LIN {X 0,Y 431.332,Z 858.27,A -85,B 0,C 180,E1 -9447.198,E2 -9447.198} C_VEL
LIN {X 0,Y 431.292,Z 859.283,A -85,B 0,C 180,E1 -9448.132,E2 -9448.132} C_VEL
LIN {X 0,Y 431.285,Z 859.901,A -85,B 0,C 180,E1 -9449.066,E2 -9449.066} C_VEL
LIN {X 0,Y 431.288,Z 860.122,A -85,B 0,C 180,E1 -9450,E2 -9450} C_VEL
LIN {X 0,Y 431.282,Z 859.894,A -85,B 0,C 180,E1 -9450.933,E2 -9450.933} C_VEL
LIN {X 0,Y 431.29,Z 859.263,A -85,B 0,C 180,E1 -9451.867,E2 -9451.867} C_VEL
LIN {X 0,Y 431.33,Z 858.237,A -85,B 0,C 180,E1 -9452.801,E2 -9452.801} C_VEL
LIN {X 0,Y 431.278,Z 856.781,A -85,B 0,C 180,E1 -9453.737,E2 -9453.737} C_VEL
LIN {X 0,Y 431.391,Z 853.758,A -85,B 0,C 180,E1 -9455.14,E2 -9455.14} C_VEL
LIN {X 0,Y 431.441,Z 849.653,A -85,B 0,C 180,E1 -9456.547,E2 -9456.547} C_VEL
LIN {X 0,Y 431.694,Z 843.326,A -85,B 0,C 180,E1 -9458.189,E2 -9458.189} C_VEL
LIN {X 0,Y 432.008,Z 836.432,A -85,B 0,C 180,E1 -9459.598,E2 -9459.598} C_VEL
LIN {X 0,Y 432.42,Z 827.793,A -85,B 0,C 180,E1 -9461.009,E2 -9461.009} C_VEL
LIN {X 0,Y 433.025,Z 818.912,A -85,B 0,C 180,E1 -9462.18,E2 -9462.18} C_VEL
LIN {X 0,Y 433.579,Z 808.605,A -85,B 0,C 180,E1 -9463.29,E2 -9463.29} C_VEL
LIN {X 0,Y 434.126,Z 798.41,A -85,B 0,C 180,E1 -9464.173,E2 -9464.173} C_VEL
LIN {X 0,Y 434.759,Z 786.373,A -85,B 0,C 180,E1 -9464.989,E2 -9464.989} C_VEL
LIN {X 0,Y 435.206,Z 773.862,A -85,B 0,C 180,E1 -9465.633,E2 -9465.633} C_VEL
LIN {X 0,Y 433.854,Z 761.171,A -85,B 0,C 180,E1 -9466.148,E2 -9466.148} C_VEL
LIN {X 0,Y 432.655,Z 748.331,A -85,B 0,C 180,E1 -9466.586,E2 -9466.586} C_VEL
LIN {X 0,Y 432.123,Z 743.343,A -85,B 0,C 180,E1 -9466.716,E2 -9466.716} C_VEL
LIN {X 0,Y 432.465,Z 730.123,A -85,B 0,C 180,E1 -9469.954,E2 -9469.954} C_VEL
LIN {X 0,Y 432.998,Z 716.144,A -85,B 0,C 180,E1 -9473.431,E2 -9473.431} C_VEL
LIN {X 0,Y 433.549,Z 704.201,A -85,B 0,C 180,E1 -9476.454,E2 -9476.454} C_VEL
LIN {X 0,Y 434.228,Z 691.104,A -85,B 0,C 180,E1 -9479.846,E2 -9479.846} C_VEL
LIN {X 0,Y 434.914,Z 679.886,A -85,B 0,C 180,E1 -9482.828,E2 -9482.828} C_VEL
LIN {X 0,Y 435.597,Z 670.042,A -85,B 0,C 180,E1 -9485.508,E2 -9485.508} C_VEL
LIN {X 0,Y 435.806,Z 664.157,A -85,B 0,C 180,E1 -9487.165,E2 -9487.165} C_VEL
LIN {X 0,Y 433.981,Z 654.686,A -85,B 0,C 180,E1 -9490.069,E2 -9490.069} C_VEL
LIN {X 0,Y 432.337,Z 646.633,A -85,B 0,C 180,E1 -9492.69,E2 -9492.69} C_VEL
LIN {X 0,Y 432.376,Z 646.627,A -85,B 0,C 180,E1 -9495.658,E2 -9495.658} C_VEL
LIN {X 0,Y 432.37,Z 646.63,A -85,B 0,C 180,E1 -9498.391,E2 -9498.391} C_VEL
LIN {X 0,Y 432.35,Z 646.63,A -85,B 0,C 180,E1 -9501.851,E2 -9501.851} C_VEL
LIN {X 0,Y 432.337,Z 646.626,A -85,B 0,C 180,E1 -9505.322,E2 -9505.322} C_VEL
LIN {X 0,Y 432.32,Z 646.63,A -85,B 0,C 180,E1 -9508.654,E2 -9508.654} C_VEL
LIN {X 0,Y 432.377,Z 646.623,A -85,B 0,C 180,E1 -9511.368,E2 -9511.368} C_VEL
LIN {X 0,Y 432.36,Z 646.625,A -85,B 0,C 180,E1 -9513.967,E2 -9513.967} C_VEL
LIN {X 0,Y 432.315,Z 646.632,A -85,B 0,C 180,E1 -9517.035,E2 -9517.035} C_VEL
LIN {X 0,Y 432.382,Z 646.622,A -85,B 0,C 180,E1 -9520.514,E2 -9520.514} C_VEL
LIN {X 0,Y 432.425,Z 646.619,A -85,B 0,C 180,E1 -9523.961,E2 -9523.961} C_VEL
LIN {X 0,Y 432.479,Z 646.612,A -85,B 0,C 180,E1 -9527.804,E2 -9527.804} C_VEL
LIN {X 0,Y 432.487,Z 646.612,A -85,B 0,C 180,E1 -9531.59,E2 -9531.59} C_VEL
LIN {X 0,Y 432.592,Z 646.601,A -85,B 0,C 180,E1 -9534.406,E2 -9534.406} C_VEL
LIN {X 0,Y 432.6,Z 646.601,A -85,B 0,C 180,E1 -9538.138,E2 -9538.138} C_VEL
LIN {X 0,Y 432.728,Z 646.587,A -85,B 0,C 180,E1 -9540,E2 -9540} C_VEL
LIN {X 0,Y 432.628,Z 646.804,A -85,B 0,C 180,E1 -9541.745,E2 -9541.745} C_VEL
LIN {X 0,Y 433.797,Z 653.829,A -85,B 0,C 180,E1 -9543.715,E2 -9543.715} C_VEL
LIN {X 0,Y 434.292,Z 658.876,A -85,B 0,C 180,E1 -9545.106,E2 -9545.106} C_VEL
LIN {X 0,Y 434.227,Z 669.203,A -85,B 0,C 180,E1 -9547.907,E2 -9547.907} C_VEL
LIN {X 0,Y 433.886,Z 681.206,A -85,B 0,C 180,E1 -9551.208,E2 -9551.208} C_VEL
LIN {X 0,Y 433.688,Z 689.494,A -85,B 0,C 180,E1 -9553.518,E2 -9553.518} C_VEL
LIN {X 0,Y 433.356,Z 701.793,A -85,B 0,C 180,E1 -9556.973,E2 -9556.973} C_VEL
LIN {X 0,Y 432.958,Z 714.047,A -85,B 0,C 180,E1 -9560.426,E2 -9560.426} C_VEL
LIN {X 0,Y 432.639,Z 724.66,A -85,B 0,C 180,E1 -9563.452,E2 -9563.452} C_VEL
LIN {X 0,Y 432.569,Z 727.887,A -85,B 0,C 180,E1 -9564.347,E2 -9564.347} C_VEL
LIN {X 0,Y 435.121,Z 741.11,A -85,B 0,C 180,E1 -9564.813,E2 -9564.813} C_VEL
LIN {X 0,Y 436.013,Z 747.455,A -85,B 0,C 180,E1 -9565.096,E2 -9565.096} C_VEL
LIN {X 0,Y 435.532,Z 759.628,A -85,B 0,C 180,E1 -9565.688,E2 -9565.688} C_VEL
LIN {X 0,Y 434.958,Z 770.483,A -85,B 0,C 180,E1 -9566.381,E2 -9566.381} C_VEL
LIN {X 0,Y 434.33,Z 781.467,A -85,B 0,C 180,E1 -9567.274,E2 -9567.274} C_VEL
LIN {X 0,Y 433.618,Z 792.684,A -85,B 0,C 180,E1 -9568.426,E2 -9568.426} C_VEL
LIN {X 0,Y 432.951,Z 802.445,A -85,B 0,C 180,E1 -9569.676,E2 -9569.676} C_VEL
LIN {X 0,Y 432.398,Z 811.473,A -85,B 0,C 180,E1 -9571.131,E2 -9571.131} C_VEL
LIN {X 0,Y 431.992,Z 818.185,A -85,B 0,C 180,E1 -9572.471,E2 -9572.471} C_VEL
LIN {X 0,Y 431.665,Z 823.82,A -85,B 0,C 180,E1 -9573.868,E2 -9573.868} C_VEL
LIN {X 0,Y 431.389,Z 828.739,A -85,B 0,C 180,E1 -9575.456,E2 -9575.456} C_VEL
LIN {X 0,Y 431.212,Z 832.39,A -85,B 0,C 180,E1 -9577.088,E2 -9577.088} C_VEL
LIN {X 0,Y 431.094,Z 834.505,A -85,B 0,C 180,E1 -9578.509,E2 -9578.509} C_VEL
LIN {X 0,Y 431.026,Z 835.696,A -85,B 0,C 180,E1 -9579.974,E2 -9579.974} C_VEL
LIN {X 0,Y 430.985,Z 835.911,A -85,B 0,C 180,E1 -9581.401,E2 -9581.401} C_VEL
LIN {X 0,Y 431.012,Z 834.855,A -85,B 0,C 180,E1 -9583.223,E2 -9583.223} C_VEL
LIN {X 0,Y 431.127,Z 833.155,A -85,B 0,C 180,E1 -9584.504,E2 -9584.504} C_VEL
LIN {X 0,Y 431.238,Z 830.613,A -85,B 0,C 180,E1 -9585.814,E2 -9585.814} C_VEL
LIN {X 0,Y 431.432,Z 827.136,A -85,B 0,C 180,E1 -9587.142,E2 -9587.142} C_VEL
LIN {X 0,Y 431.652,Z 822.558,A -85,B 0,C 180,E1 -9588.5,E2 -9588.5} C_VEL
LIN {X 0,Y 431.99,Z 816.732,A -85,B 0,C 180,E1 -9589.875,E2 -9589.875} C_VEL
LIN {X 0,Y 432.47,Z 809.427,A -85,B 0,C 180,E1 -9591.264,E2 -9591.264} C_VEL
LIN {X 0,Y 432.989,Z 801.184,A -85,B 0,C 180,E1 -9592.533,E2 -9592.533} C_VEL
LIN {X 0,Y 433.608,Z 791.196,A -85,B 0,C 180,E1 -9593.776,E2 -9593.776} C_VEL
LIN {X 0,Y 434.236,Z 781.145,A -85,B 0,C 180,E1 -9594.791,E2 -9594.791} C_VEL
LIN {X 0,Y 434.882,Z 769.922,A -85,B 0,C 180,E1 -9595.695,E2 -9595.695} C_VEL
LIN {X 0,Y 435.548,Z 757.776,A -85,B 0,C 180,E1 -9596.451,E2 -9596.451} C_VEL
LIN {X 0,Y 435.872,Z 746.742,A -85,B 0,C 180,E1 -9596.977,E2 -9596.977} C_VEL
LIN {X 0,Y 433.746,Z 734.023,A -85,B 0,C 180,E1 -9597.492,E2 -9597.492} C_VEL
LIN {X 0,Y 432.461,Z 727.38,A -85,B 0,C 180,E1 -9597.714,E2 -9597.714} C_VEL
LIN {X 0,Y 432.921,Z 715.217,A -85,B 0,C 180,E1 -9601.238,E2 -9601.238} C_VEL
LIN {X 0,Y 433.297,Z 703.777,A -85,B 0,C 180,E1 -9604.544,E2 -9604.544} C_VEL
LIN {X 0,Y 433.675,Z 692.539,A -85,B 0,C 180,E1 -9607.802,E2 -9607.802} C_VEL
LIN {X 0,Y 434.013,Z 682.851,A -85,B 0,C 180,E1 -9610.613,E2 -9610.613} C_VEL
LIN {X 0,Y 434.368,Z 671.056,A -85,B 0,C 180,E1 -9614.035,E2 -9614.035} C_VEL
LIN {X 0,Y 434.561,Z 661.142,A -85,B 0,C 180,E1 -9616.914,E2 -9616.914} C_VEL
LIN {X 0,Y 434.514,Z 659.446,A -85,B 0,C 180,E1 -9617.42,E2 -9617.42} C_VEL
LIN {X 0,Y 433.592,Z 657.241,A -85,B 0,C 180,E1 -9618.132,E2 -9618.132} C_VEL
LIN {X 0,Y 430.211,Z 654.112,A -85,B 0,C 180,E1 -9619.298,E2 -9619.298} C_VEL
LIN {X 0,Y 427.311,Z 651.652,A -85,B 0,C 180,E1 -9620.24,E2 -9620.24} C_VEL
LIN {X 0,Y 425.886,Z 649.565,A -85,B 0,C 180,E1 -9620.965,E2 -9620.965} C_VEL
LIN {X 0,Y 425.67,Z 648.783,A -85,B 0,C 180,E1 -9621.21,E2 -9621.21} C_VEL
LIN {X 0,Y 425.459,Z 647.491,A -85,B 0,C 180,E1 -9621.63,E2 -9621.63} C_VEL
LIN {X 0,Y 425.555,Z 647.481,A -85,B 0,C 180,E1 -9624.314,E2 -9624.314} C_VEL
LIN {X 0,Y 425.577,Z 647.478,A -85,B 0,C 180,E1 -9628.108,E2 -9628.108} C_VEL
LIN {X 0,Y 425.705,Z 647.459,A -85,B 0,C 180,E1 -9630.001,E2 -9630.001} C_VEL
LIN {X 0,Y 425.559,Z 647.477,A -85,B 0,C 180,E1 -9632.84,E2 -9632.84} C_VEL
LIN {X 0,Y 425.528,Z 647.477,A -85,B 0,C 180,E1 -9636.639,E2 -9636.639} C_VEL
LIN {X 0,Y 425.405,Z 647.493,A -85,B 0,C 180,E1 -9639.51,E2 -9639.51} C_VEL
LIN {X 0,Y 425.406,Z 647.497,A -85,B 0,C 180,E1 -9642.911,E2 -9642.911} C_VEL
LIN {X 0,Y 425.363,Z 647.504,A -85,B 0,C 180,E1 -9646.605,E2 -9646.605} C_VEL
LIN {X 0,Y 425.33,Z 647.508,A -85,B 0,C 180,E1 -9649.636,E2 -9649.636} C_VEL
LIN {X 0,Y 425.334,Z 647.574,A -85,B 0,C 180,E1 -9651.996,E2 -9651.996} C_VEL
LIN {X 0,Y 428.652,Z 658.894,A -85,B 0,C 180,E1 -9652.79,E2 -9652.79} C_VEL
LIN {X 0,Y 429.276,Z 661.664,A -85,B 0,C 180,E1 -9653.009,E2 -9653.009} C_VEL
LIN {X 0,Y 428.845,Z 672.85,A -85,B 0,C 180,E1 -9653.875,E2 -9653.875} C_VEL
LIN {X 0,Y 428.275,Z 683.125,A -85,B 0,C 180,E1 -9654.867,E2 -9654.867} C_VEL
LIN {X 0,Y 427.705,Z 693.237,A -85,B 0,C 180,E1 -9656.087,E2 -9656.087} C_VEL
LIN {X 0,Y 427.131,Z 702.284,A -85,B 0,C 180,E1 -9657.433,E2 -9657.433} C_VEL
LIN {X 0,Y 426.579,Z 709.888,A -85,B 0,C 180,E1 -9658.839,E2 -9658.839} C_VEL
LIN {X 0,Y 426.091,Z 716.875,A -85,B 0,C 180,E1 -9660.477,E2 -9660.477} C_VEL
LIN {X 0,Y 425.795,Z 721.556,A -85,B 0,C 180,E1 -9661.883,E2 -9661.883} C_VEL
LIN {X 0,Y 425.508,Z 725.849,A -85,B 0,C 180,E1 -9663.595,E2 -9663.595} C_VEL
LIN {X 0,Y 425.268,Z 728.728,A -85,B 0,C 180,E1 -9665.339,E2 -9665.339} C_VEL
LIN {X 0,Y 425.19,Z 729.934,A -85,B 0,C 180,E1 -9666.516,E2 -9666.516} C_VEL
LIN {X 0,Y 425.178,Z 730.484,A -85,B 0,C 180,E1 -9667.705,E2 -9667.705} C_VEL
LIN {X 0,Y 425.238,Z 730.406,A -85,B 0,C 180,E1 -9669.033,E2 -9669.033} C_VEL
LIN {X 0,Y 425.33,Z 729.404,A -85,B 0,C 180,E1 -9670.528,E2 -9670.528} C_VEL
LIN {X 0,Y 425.479,Z 727.476,A -85,B 0,C 180,E1 -9671.987,E2 -9671.987} C_VEL
LIN {X 0,Y 425.747,Z 724.603,A -85,B 0,C 180,E1 -9673.421,E2 -9673.421} C_VEL
LIN {X 0,Y 426.153,Z 719.68,A -85,B 0,C 180,E1 -9675.166,E2 -9675.166} C_VEL
LIN {X 0,Y 426.643,Z 713.798,A -85,B 0,C 180,E1 -9676.735,E2 -9676.735} C_VEL
LIN {X 0,Y 427.105,Z 707.513,A -85,B 0,C 180,E1 -9678.061,E2 -9678.061} C_VEL
LIN {X 0,Y 427.71,Z 699.733,A -85,B 0,C 180,E1 -9679.387,E2 -9679.387} C_VEL
LIN {X 0,Y 428.308,Z 691.12,A -85,B 0,C 180,E1 -9680.585,E2 -9680.585} C_VEL
LIN {X 0,Y 428.931,Z 681.12,A -85,B 0,C 180,E1 -9681.717,E2 -9681.717} C_VEL
LIN {X 0,Y 429.438,Z 671.625,A -85,B 0,C 180,E1 -9682.589,E2 -9682.589} C_VEL
LIN {X 0,Y 429.657,Z 661.647,A -85,B 0,C 180,E1 -9683.341,E2 -9683.341} C_VEL
LIN {X 0,Y 426.566,Z 651.552,A -85,B 0,C 180,E1 -9684.105,E2 -9684.105} C_VEL
LIN {X 0,Y 425.297,Z 647.508,A -85,B 0,C 180,E1 -9684.371,E2 -9684.371} C_VEL
LIN {X 0,Y 425.282,Z 647.515,A -85,B 0,C 180,E1 -9687.437,E2 -9687.437} C_VEL
LIN {X 0,Y 425.292,Z 647.507,A -85,B 0,C 180,E1 -9690.281,E2 -9690.281} C_VEL
LIN {X 0,Y 425.354,Z 647.499,A -85,B 0,C 180,E1 -9693.506,E2 -9693.506} C_VEL
LIN {X 0,Y 425.285,Z 647.502,A -85,B 0,C 180,E1 -9696.634,E2 -9696.634} C_VEL
LIN {X 0,Y 425.296,Z 647.513,A -85,B 0,C 180,E1 -9699.695,E2 -9699.695} C_VEL
LIN {X 0,Y 425.344,Z 647.499,A -85,B 0,C 180,E1 -9702.698,E2 -9702.698} C_VEL
LIN {X 0,Y 425.352,Z 647.503,A -85,B 0,C 180,E1 -9705.65,E2 -9705.65} C_VEL
LIN {X 0,Y 425.352,Z 647.496,A -85,B 0,C 180,E1 -9708.564,E2 -9708.564} C_VEL
LIN {X 0,Y 425.539,Z 647.472,A -85,B 0,C 180,E1 -9712.408,E2 -9712.408} C_VEL
LIN {X 0,Y 425.555,Z 647.476,A -85,B 0,C 180,E1 -9714.313,E2 -9714.313} C_VEL
LIN {X 0,Y 425.577,Z 647.474,A -85,B 0,C 180,E1 -9718.107,E2 -9718.107} C_VEL
LIN {X 0,Y 425.705,Z 647.455,A -85,B 0,C 180,E1 -9720,E2 -9720} C_VEL
LIN {X 0,Y 425.559,Z 647.472,A -85,B 0,C 180,E1 -9722.84,E2 -9722.84} C_VEL
LIN {X 0,Y 425.532,Z 647.478,A -85,B 0,C 180,E1 -9726.639,E2 -9726.639} C_VEL
LIN {X 0,Y 425.403,Z 647.487,A -85,B 0,C 180,E1 -9729.509,E2 -9729.509} C_VEL
LIN {X 0,Y 425.395,Z 647.49,A -85,B 0,C 180,E1 -9732.904,E2 -9732.904} C_VEL
LIN {X 0,Y 425.363,Z 647.497,A -85,B 0,C 180,E1 -9736.605,E2 -9736.605} C_VEL
LIN {X 0,Y 425.33,Z 647.5,A -85,B 0,C 180,E1 -9739.636,E2 -9739.636} C_VEL
LIN {X 0,Y 425.309,Z 647.502,A -85,B 0,C 180,E1 -9743.365,E2 -9743.365} C_VEL
LIN {X 0,Y 425.349,Z 647.502,A -85,B 0,C 180,E1 -9746.844,E2 -9746.844} C_VEL
LIN {X 0,Y 425.293,Z 647.507,A -85,B 0,C 180,E1 -9749.72,E2 -9749.72} C_VEL
LIN {X 0,Y 425.284,Z 647.511,A -85,B 0,C 180,E1 -9753.048,E2 -9753.048} C_VEL
LIN {X 0,Y 425.284,Z 647.511,A -85,B 0,C 180,E1 -9755.929,E2 -9755.929} C_VEL
LIN {X 0,Y 425.296,Z 647.511,A -85,B 0,C 180,E1 -9759.043,E2 -9759.043} C_VEL
LIN {X 0,Y 425.277,Z 647.51,A -85,B 0,C 180,E1 -9762.653,E2 -9762.653} C_VEL
LIN {X 0,Y 425.264,Z 647.515,A -85,B 0,C 180,E1 -9766.044,E2 -9766.044} C_VEL
LIN {X 0,Y 425.339,Z 647.645,A -85,B 0,C 180,E1 -9767.56,E2 -9767.56} C_VEL
LIN {X 0,Y 427.156,Z 656.735,A -85,B 0,C 180,E1 -9770.651,E2 -9770.651} C_VEL
LIN {X 0,Y 428.474,Z 664.587,A -85,B 0,C 180,E1 -9773.118,E2 -9773.118} C_VEL
LIN {X 0,Y 428.013,Z 671.749,A -85,B 0,C 180,E1 -9775.186,E2 -9775.186} C_VEL
LIN {X 0,Y 427.234,Z 684.05,A -85,B 0,C 180,E1 -9778.579,E2 -9778.579} C_VEL
LIN {X 0,Y 426.511,Z 697.918,A -85,B 0,C 180,E1 -9782.257,E2 -9782.257} C_VEL
LIN {X 0,Y 425.939,Z 711.089,A -85,B 0,C 180,E1 -9785.638,E2 -9785.638} C_VEL
LIN {X 0,Y 425.433,Z 724.268,A -85,B 0,C 180,E1 -9788.942,E2 -9788.942} C_VEL
LIN {X 0,Y 425.109,Z 737.422,A -85,B 0,C 180,E1 -9792.191,E2 -9792.191} C_VEL
LIN {X 0,Y 425.001,Z 740.706,A -85,B 0,C 180,E1 -9792.945,E2 -9792.945} C_VEL
LIN {X 0,Y 426.386,Z 753.802,A -85,B 0,C 180,E1 -9793.347,E2 -9793.347} C_VEL
LIN {X 0,Y 427.922,Z 771.686,A -85,B 0,C 180,E1 -9794.047,E2 -9794.047} C_VEL
LIN {X 0,Y 428.234,Z 776.777,A -85,B 0,C 180,E1 -9794.288,E2 -9794.288} C_VEL
LIN {X 0,Y 427.815,Z 787.707,A -85,B 0,C 180,E1 -9794.883,E2 -9794.883} C_VEL
LIN {X 0,Y 427.112,Z 799.468,A -85,B 0,C 180,E1 -9795.71,E2 -9795.71} C_VEL
LIN {X 0,Y 426.476,Z 811.174,A -85,B 0,C 180,E1 -9796.782,E2 -9796.782} C_VEL
LIN {X 0,Y 425.94,Z 820.608,A -85,B 0,C 180,E1 -9797.855,E2 -9797.855} C_VEL
LIN {X 0,Y 425.369,Z 829.198,A -85,B 0,C 180,E1 -9799.047,E2 -9799.047} C_VEL
LIN {X 0,Y 424.891,Z 837.512,A -85,B 0,C 180,E1 -9800.479,E2 -9800.479} C_VEL
LIN {X 0,Y 424.585,Z 844.19,A -85,B 0,C 180,E1 -9801.911,E2 -9801.911} C_VEL
LIN {X 0,Y 424.378,Z 850.124,A -85,B 0,C 180,E1 -9803.538,E2 -9803.538} C_VEL
LIN {X 0,Y 424.29,Z 854.698,A -85,B 0,C 180,E1 -9805.249,E2 -9805.249} C_VEL
LIN {X 0,Y 424.192,Z 856.61,A -85,B 0,C 180,E1 -9806.2,E2 -9806.2} C_VEL
LIN {X 0,Y 424.228,Z 858.067,A -85,B 0,C 180,E1 -9807.151,E2 -9807.151} C_VEL
LIN {X 0,Y 424.214,Z 859.082,A -85,B 0,C 180,E1 -9808.101,E2 -9808.101} C_VEL
LIN {X 0,Y 424.199,Z 859.701,A -85,B 0,C 180,E1 -9809.05,E2 -9809.05} C_VEL
LIN {X 0,Y 424.198,Z 859.923,A -85,B 0,C 180,E1 -9809.999,E2 -9809.999} C_VEL
LIN {X 0,Y 424.195,Z 859.696,A -85,B 0,C 180,E1 -9810.949,E2 -9810.949} C_VEL
LIN {X 0,Y 424.212,Z 859.066,A -85,B 0,C 180,E1 -9811.898,E2 -9811.898} C_VEL
LIN {X 0,Y 424.226,Z 858.04,A -85,B 0,C 180,E1 -9812.848,E2 -9812.848} C_VEL
LIN {X 0,Y 424.185,Z 856.587,A -85,B 0,C 180,E1 -9813.799,E2 -9813.799} C_VEL
LIN {X 0,Y 424.301,Z 853.567,A -85,B 0,C 180,E1 -9815.226,E2 -9815.226} C_VEL
LIN {X 0,Y 424.359,Z 849.468,A -85,B 0,C 180,E1 -9816.657,E2 -9816.657} C_VEL
LIN {X 0,Y 424.629,Z 843.148,A -85,B 0,C 180,E1 -9818.326,E2 -9818.326} C_VEL
LIN {X 0,Y 424.974,Z 836.256,A -85,B 0,C 180,E1 -9819.759,E2 -9819.759} C_VEL
LIN {X 0,Y 425.426,Z 827.626,A -85,B 0,C 180,E1 -9821.192,E2 -9821.192} C_VEL
LIN {X 0,Y 426.053,Z 818.752,A -85,B 0,C 180,E1 -9822.382,E2 -9822.382} C_VEL
LIN {X 0,Y 426.662,Z 808.119,A -85,B 0,C 180,E1 -9823.544,E2 -9823.544} C_VEL
LIN {X 0,Y 427.315,Z 796.719,A -85,B 0,C 180,E1 -9824.525,E2 -9824.525} C_VEL
LIN {X 0,Y 428.016,Z 784.329,A -85,B 0,C 180,E1 -9825.353,E2 -9825.353} C_VEL
LIN {X 0,Y 428.22,Z 773.834,A -85,B 0,C 180,E1 -9825.894,E2 -9825.894} C_VEL
LIN {X 0,Y 427.029,Z 761.62,A -85,B 0,C 180,E1 -9826.407,E2 -9826.407} C_VEL
LIN {X 0,Y 425.059,Z 742.377,A -85,B 0,C 180,E1 -9826.992,E2 -9826.992} C_VEL
LIN {X 0,Y 425.44,Z 729.173,A -85,B 0,C 180,E1 -9830.298,E2 -9830.298} C_VEL
LIN {X 0,Y 425.896,Z 717.225,A -85,B 0,C 180,E1 -9833.33,E2 -9833.33} C_VEL
LIN {X 0,Y 426.477,Z 705.265,A -85,B 0,C 180,E1 -9836.419,E2 -9836.419} C_VEL
LIN {X 0,Y 427.207,Z 692.269,A -85,B 0,C 180,E1 -9839.843,E2 -9839.843} C_VEL
LIN {X 0,Y 427.898,Z 681.246,A -85,B 0,C 180,E1 -9842.82,E2 -9842.82} C_VEL
LIN {X 0,Y 428.699,Z 670.246,A -85,B 0,C 180,E1 -9845.878,E2 -9845.878} C_VEL
LIN {X 0,Y 428.812,Z 665.206,A -85,B 0,C 180,E1 -9847.329,E2 -9847.329} C_VEL
LIN {X 0,Y 426.954,Z 655.628,A -85,B 0,C 180,E1 -9850.327,E2 -9850.327} C_VEL
LIN {X 0,Y 425.296,Z 647.51,A -85,B 0,C 180,E1 -9853.023,E2 -9853.023} C_VEL
LIN {X 0,Y 425.329,Z 647.508,A -85,B 0,C 180,E1 -9856.638,E2 -9856.638} C_VEL
LIN {X 0,Y 425.309,Z 647.507,A -85,B 0,C 180,E1 -9859.875,E2 -9859.875} C_VEL
LIN {X 0,Y 425.284,Z 647.507,A -85,B 0,C 180,E1 -9862.486,E2 -9862.486} C_VEL
LIN {X 0,Y 425.304,Z 647.504,A -85,B 0,C 180,E1 -9865.817,E2 -9865.817} C_VEL
LIN {X 0,Y 425.296,Z 647.505,A -85,B 0,C 180,E1 -9869.236,E2 -9869.236} C_VEL
LIN {X 0,Y 425.346,Z 647.501,A -85,B 0,C 180,E1 -9872.442,E2 -9872.442} C_VEL
LIN {X 0,Y 425.347,Z 647.505,A -85,B 0,C 180,E1 -9875.602,E2 -9875.602} C_VEL
LIN {X 0,Y 425.288,Z 647.509,A -85,B 0,C 180,E1 -9878.681,E2 -9878.681} C_VEL
LIN {X 0,Y 425.328,Z 647.502,A -85,B 0,C 180,E1 -9881.702,E2 -9881.702} C_VEL
LIN {X 0,Y 425.344,Z 647.502,A -85,B 0,C 180,E1 -9884.67,E2 -9884.67} C_VEL
LIN {X 0,Y 425.427,Z 647.492,A -85,B 0,C 180,E1 -9887.598,E2 -9887.598} C_VEL
LIN {X 0,Y 425.438,Z 647.491,A -85,B 0,C 180,E1 -9891.45,E2 -9891.45} C_VEL
LIN {X 0,Y 425.549,Z 647.479,A -85,B 0,C 180,E1 -9894.313,E2 -9894.313} C_VEL
LIN {X 0,Y 425.57,Z 647.477,A -85,B 0,C 180,E1 -9898.107,E2 -9898.107} C_VEL
LIN {X 0,Y 425.697,Z 647.463,A -85,B 0,C 180,E1 -9900,E2 -9900} C_VEL
LIN {X 0,Y 425.55,Z 647.558,A -85,B 0,C 180,E1 -9901.36,E2 -9901.36} C_VEL
LIN {X 0,Y 426.769,Z 654.365,A -85,B 0,C 180,E1 -9903.304,E2 -9903.304} C_VEL
LIN {X 0,Y 427.351,Z 659.35,A -85,B 0,C 180,E1 -9904.716,E2 -9904.716} C_VEL
LIN {X 0,Y 427.342,Z 669.736,A -85,B 0,C 180,E1 -9907.56,E2 -9907.56} C_VEL
LIN {X 0,Y 426.974,Z 680.051,A -85,B 0,C 180,E1 -9910.431,E2 -9910.431} C_VEL
LIN {X 0,Y 426.809,Z 688.62,A -85,B 0,C 180,E1 -9912.844,E2 -9912.844} C_VEL
LIN {X 0,Y 426.477,Z 699.066,A -85,B 0,C 180,E1 -9915.778,E2 -9915.778} C_VEL
LIN {X 0,Y 426.153,Z 709.567,A -85,B 0,C 180,E1 -9918.759,E2 -9918.759} C_VEL
LIN {X 0,Y 425.82,Z 720.147,A -85,B 0,C 180,E1 -9921.799,E2 -9921.799} C_VEL
LIN {X 0,Y 425.592,Z 727.868,A -85,B 0,C 180,E1 -9924.026,E2 -9924.026} C_VEL
LIN {X 0,Y 428.378,Z 742.541,A -85,B 0,C 180,E1 -9924.587,E2 -9924.587} C_VEL
LIN {X 0,Y 429.178,Z 749.058,A -85,B 0,C 180,E1 -9924.89,E2 -9924.89} C_VEL
LIN {X 0,Y 428.69,Z 760.796,A -85,B 0,C 180,E1 -9925.487,E2 -9925.487} C_VEL
LIN {X 0,Y 428.07,Z 771.625,A -85,B 0,C 180,E1 -9926.205,E2 -9926.205} C_VEL
LIN {X 0,Y 427.389,Z 782.348,A -85,B 0,C 180,E1 -9927.107,E2 -9927.107} C_VEL
LIN {X 0,Y 426.65,Z 793.363,A -85,B 0,C 180,E1 -9928.267,E2 -9928.267} C_VEL
LIN {X 0,Y 425.972,Z 802.787,A -85,B 0,C 180,E1 -9929.503,E2 -9929.503} C_VEL
LIN {X 0,Y 425.447,Z 810.807,A -85,B 0,C 180,E1 -9930.803,E2 -9930.803} C_VEL
LIN {X 0,Y 425.006,Z 817.896,A -85,B 0,C 180,E1 -9932.215,E2 -9932.215} C_VEL
LIN {X 0,Y 424.651,Z 823.543,A -85,B 0,C 180,E1 -9933.611,E2 -9933.611} C_VEL
LIN {X 0,Y 424.305,Z 829.136,A -85,B 0,C 180,E1 -9935.431,E2 -9935.431} C_VEL
LIN {X 0,Y 424.183,Z 831.864,A -85,B 0,C 180,E1 -9936.617,E2 -9936.617} C_VEL
LIN {X 0,Y 424.075,Z 833.895,A -85,B 0,C 180,E1 -9937.82,E2 -9937.82} C_VEL
LIN {X 0,Y 423.95,Z 835.297,A -85,B 0,C 180,E1 -9939.046,E2 -9939.046} C_VEL
LIN {X 0,Y 423.919,Z 836.06,A -85,B 0,C 180,E1 -9940.306,E2 -9940.306} C_VEL
LIN {X 0,Y 423.901,Z 836.045,A -85,B 0,C 180,E1 -9941.75,E2 -9941.75} C_VEL
LIN {X 0,Y 423.911,Z 835.132,A -85,B 0,C 180,E1 -9943.159,E2 -9943.159} C_VEL
LIN {X 0,Y 424.034,Z 833.36,A -85,B 0,C 180,E1 -9944.547,E2 -9944.547} C_VEL
LIN {X 0,Y 424.157,Z 830.768,A -85,B 0,C 180,E1 -9945.901,E2 -9945.901} C_VEL
LIN {X 0,Y 424.358,Z 827.326,A -85,B 0,C 180,E1 -9947.234,E2 -9947.234} C_VEL
LIN {X 0,Y 424.653,Z 822,A -85,B 0,C 180,E1 -9948.812,E2 -9948.812} C_VEL
LIN {X 0,Y 425.074,Z 814.92,A -85,B 0,C 180,E1 -9950.427,E2 -9950.427} C_VEL
LIN {X 0,Y 425.548,Z 807.735,A -85,B 0,C 180,E1 -9951.735,E2 -9951.735} C_VEL
LIN {X 0,Y 426.221,Z 798.161,A -85,B 0,C 180,E1 -9953.146,E2 -9953.146} C_VEL
LIN {X 0,Y 426.953,Z 787.532,A -85,B 0,C 180,E1 -9954.388,E2 -9954.388} C_VEL
LIN {X 0,Y 427.594,Z 777.252,A -85,B 0,C 180,E1 -9955.359,E2 -9955.359} C_VEL
LIN {X 0,Y 428.225,Z 766.551,A -85,B 0,C 180,E1 -9956.169,E2 -9956.169} C_VEL
LIN {X 0,Y 428.837,Z 753.63,A -85,B 0,C 180,E1 -9956.915,E2 -9956.915} C_VEL
LIN {X 0,Y 429.043,Z 747.886,A -85,B 0,C 180,E1 -9957.179,E2 -9957.179} C_VEL
LIN {X 0,Y 426.915,Z 735.03,A -85,B 0,C 180,E1 -9957.726,E2 -9957.726} C_VEL
LIN {X 0,Y 425.485,Z 727.51,A -85,B 0,C 180,E1 -9957.982,E2 -9957.982} C_VEL
LIN {X 0,Y 425.916,Z 715.771,A -85,B 0,C 180,E1 -9961.412,E2 -9961.412} C_VEL
LIN {X 0,Y 426.3,Z 704.802,A -85,B 0,C 180,E1 -9964.62,E2 -9964.62} C_VEL
LIN {X 0,Y 426.672,Z 694.137,A -85,B 0,C 180,E1 -9967.738,E2 -9967.738} C_VEL
LIN {X 0,Y 427.055,Z 683.725,A -85,B 0,C 180,E1 -9970.784,E2 -9970.784} C_VEL
LIN {X 0,Y 427.437,Z 671.868,A -85,B 0,C 180,E1 -9974.259,E2 -9974.259} C_VEL
LIN {X 0,Y 427.626,Z 661.902,A -85,B 0,C 180,E1 -9977.182,E2 -9977.182} C_VEL
LIN {X 0,Y 426.933,Z 655.631,A -85,B 0,C 180,E1 -9979.088,E2 -9979.088} C_VEL
LIN {X 0,Y 425.67,Z 648.783,A -85,B 0,C 180,E1 -9981.21,E2 -9981.21} C_VEL
LIN {X 0,Y 425.132,Z 647.83,A -85,B 0,C 180,E1 -9981.703,E2 -9981.703} C_VEL
LIN {X 0,Y 424.201,Z 647.646,A -85,B 0,C 180,E1 -9982.211,E2 -9982.211} C_VEL
LIN {X 0,Y 419.432,Z 648.323,A -85,B 0,C 180,E1 -9984.292,E2 -9984.292} C_VEL
LIN {X 0,Y 418.42,Z 648.379,A -85,B 0,C 180,E1 -9985.109,E2 -9985.109} C_VEL
LIN {X 0,Y 418.322,Z 648.381,A -85,B 0,C 180,E1 -9985.385,E2 -9985.385} C_VEL
LIN {X 0,Y 418.546,Z 648.353,A -85,B 0,C 180,E1 -9988.076,E2 -9988.076} C_VEL
LIN {X 0,Y 418.674,Z 648.335,A -85,B 0,C 180,E1 -9990.001,E2 -9990.001} C_VEL
LIN {X 0,Y 418.513,Z 648.354,A -85,B 0,C 180,E1 -9992.888,E2 -9992.888} C_VEL
LIN {X 0,Y 418.492,Z 648.353,A -85,B 0,C 180,E1 -9996.752,E2 -9996.752} C_VEL
LIN {X 0,Y 418.361,Z 648.37,A -85,B 0,C 180,E1 -9999.671,E2 -9999.671} C_VEL
LIN {X 0,Y 418.357,Z 648.374,A -85,B 0,C 180,E1 -10003.007,E2 -10003.007} C_VEL
LIN {X 0,Y 418.315,Z 648.381,A -85,B 0,C 180,E1 -10006.736,E2 -10006.736} C_VEL
LIN {X 0,Y 418.284,Z 648.385,A -85,B 0,C 180,E1 -10009.795,E2 -10009.795} C_VEL
LIN {X 0,Y 418.307,Z 648.382,A -85,B 0,C 180,E1 -10011.72,E2 -10011.72} C_VEL
LIN {X 0,Y 421.639,Z 659.821,A -85,B 0,C 180,E1 -10012.543,E2 -10012.543} C_VEL
LIN {X 0,Y 422.388,Z 662.544,A -85,B 0,C 180,E1 -10012.768,E2 -10012.768} C_VEL
LIN {X 0,Y 422.006,Z 673.831,A -85,B 0,C 180,E1 -10013.658,E2 -10013.658} C_VEL
LIN {X 0,Y 421.425,Z 683.885,A -85,B 0,C 180,E1 -10014.641,E2 -10014.641} C_VEL
LIN {X 0,Y 420.841,Z 693.947,A -85,B 0,C 180,E1 -10015.867,E2 -10015.867} C_VEL
LIN {X 0,Y 420.266,Z 702.746,A -85,B 0,C 180,E1 -10017.187,E2 -10017.187} C_VEL
LIN {X 0,Y 419.691,Z 709.946,A -85,B 0,C 180,E1 -10018.506,E2 -10018.506} C_VEL
LIN {X 0,Y 419.304,Z 715.451,A -85,B 0,C 180,E1 -10019.739,E2 -10019.739} C_VEL
LIN {X 0,Y 418.892,Z 721.217,A -85,B 0,C 180,E1 -10021.34,E2 -10021.34} C_VEL
LIN {X 0,Y 418.594,Z 725.495,A -85,B 0,C 180,E1 -10022.915,E2 -10022.915} C_VEL
LIN {X 0,Y 418.298,Z 729.122,A -85,B 0,C 180,E1 -10024.838,E2 -10024.838} C_VEL
LIN {X 0,Y 418.177,Z 730.71,A -85,B 0,C 180,E1 -10026.225,E2 -10026.225} C_VEL
LIN {X 0,Y 418.154,Z 731.535,A -85,B 0,C 180,E1 -10027.82,E2 -10027.82} C_VEL
LIN {X 0,Y 418.246,Z 731.163,A -85,B 0,C 180,E1 -10029.683,E2 -10029.683} C_VEL
LIN {X 0,Y 418.361,Z 730.067,A -85,B 0,C 180,E1 -10030.932,E2 -10030.932} C_VEL
LIN {X 0,Y 418.637,Z 727.035,A -85,B 0,C 180,E1 -10032.876,E2 -10032.876} C_VEL
LIN {X 0,Y 418.953,Z 723.836,A -85,B 0,C 180,E1 -10034.248,E2 -10034.248} C_VEL
LIN {X 0,Y 419.313,Z 719.692,A -85,B 0,C 180,E1 -10035.616,E2 -10035.616} C_VEL
LIN {X 0,Y 419.754,Z 714.49,A -85,B 0,C 180,E1 -10036.977,E2 -10036.977} C_VEL
LIN {X 0,Y 420.326,Z 706.835,A -85,B 0,C 180,E1 -10038.563,E2 -10038.563} C_VEL
LIN {X 0,Y 420.933,Z 699.393,A -85,B 0,C 180,E1 -10039.804,E2 -10039.804} C_VEL
LIN {X 0,Y 421.536,Z 691.319,A -85,B 0,C 180,E1 -10040.916,E2 -10040.916} C_VEL
LIN {X 0,Y 422.173,Z 681.946,A -85,B 0,C 180,E1 -10041.979,E2 -10041.979} C_VEL
LIN {X 0,Y 422.742,Z 671.495,A -85,B 0,C 180,E1 -10042.939,E2 -10042.939} C_VEL
LIN {X 0,Y 423.029,Z 663.901,A -85,B 0,C 180,E1 -10043.513,E2 -10043.513} C_VEL
LIN {X 0,Y 419.591,Z 652.47,A -85,B 0,C 180,E1 -10044.405,E2 -10044.405} C_VEL
LIN {X 0,Y 418.265,Z 648.384,A -85,B 0,C 180,E1 -10044.7,E2 -10044.7} C_VEL
LIN {X 0,Y 418.246,Z 648.392,A -85,B 0,C 180,E1 -10047.472,E2 -10047.472} C_VEL
LIN {X 0,Y 418.269,Z 648.381,A -85,B 0,C 180,E1 -10050.896,E2 -10050.896} C_VEL
LIN {X 0,Y 418.269,Z 648.382,A -85,B 0,C 180,E1 -10054.096,E2 -10054.096} C_VEL
LIN {X 0,Y 418.232,Z 648.381,A -85,B 0,C 180,E1 -10057.264,E2 -10057.264} C_VEL
LIN {X 0,Y 418.284,Z 648.382,A -85,B 0,C 180,E1 -10060.364,E2 -10060.364} C_VEL
LIN {X 0,Y 418.327,Z 648.376,A -85,B 0,C 180,E1 -10063.405,E2 -10063.405} C_VEL
LIN {X 0,Y 418.347,Z 648.372,A -85,B 0,C 180,E1 -10066.999,E2 -10066.999} C_VEL
LIN {X 0,Y 418.342,Z 648.374,A -85,B 0,C 180,E1 -10070.329,E2 -10070.329} C_VEL
LIN {X 0,Y 418.515,Z 648.348,A -85,B 0,C 180,E1 -10072.28,E2 -10072.28} C_VEL
LIN {X 0,Y 418.515,Z 648.354,A -85,B 0,C 180,E1 -10074.217,E2 -10074.217} C_VEL
LIN {X 0,Y 418.546,Z 648.349,A -85,B 0,C 180,E1 -10078.076,E2 -10078.076} C_VEL
LIN {X 0,Y 418.674,Z 648.331,A -85,B 0,C 180,E1 -10080,E2 -10080} C_VEL
LIN {X 0,Y 418.512,Z 648.35,A -85,B 0,C 180,E1 -10082.888,E2 -10082.888} C_VEL
LIN {X 0,Y 418.495,Z 648.353,A -85,B 0,C 180,E1 -10086.751,E2 -10086.751} C_VEL
LIN {X 0,Y 418.402,Z 648.36,A -85,B 0,C 180,E1 -10088.695,E2 -10088.695} C_VEL
LIN {X 0,Y 418.317,Z 648.376,A -85,B 0,C 180,E1 -10091.631,E2 -10091.631} C_VEL
LIN {X 0,Y 418.304,Z 648.38,A -85,B 0,C 180,E1 -10094.597,E2 -10094.597} C_VEL
LIN {X 0,Y 418.289,Z 648.376,A -85,B 0,C 180,E1 -10097.604,E2 -10097.604} C_VEL
LIN {X 0,Y 418.252,Z 648.387,A -85,B 0,C 180,E1 -10100.663,E2 -10100.663} C_VEL
LIN {X 0,Y 418.29,Z 648.377,A -85,B 0,C 180,E1 -10103.781,E2 -10103.781} C_VEL
LIN {X 0,Y 418.312,Z 648.377,A -85,B 0,C 180,E1 -10107.071,E2 -10107.071} C_VEL
LIN {X 0,Y 418.246,Z 648.388,A -85,B 0,C 180,E1 -10110.272,E2 -10110.272} C_VEL
LIN {X 0,Y 418.25,Z 648.385,A -85,B 0,C 180,E1 -10113.677,E2 -10113.677} C_VEL
LIN {X 0,Y 418.242,Z 648.389,A -85,B 0,C 180,E1 -10117.224,E2 -10117.224} C_VEL
LIN {X 0,Y 418.251,Z 648.386,A -85,B 0,C 180,E1 -10119.682,E2 -10119.682} C_VEL
LIN {X 0,Y 418.232,Z 648.391,A -85,B 0,C 180,E1 -10122.321,E2 -10122.321} C_VEL
LIN {X 0,Y 418.238,Z 648.391,A -85,B 0,C 180,E1 -10125.109,E2 -10125.109} C_VEL
LIN {X 0,Y 418.279,Z 648.479,A -85,B 0,C 180,E1 -10127.176,E2 -10127.176} C_VEL
LIN {X 0,Y 420.089,Z 657.482,A -85,B 0,C 180,E1 -10130.316,E2 -10130.316} C_VEL
LIN {X 0,Y 421.435,Z 665.136,A -85,B 0,C 180,E1 -10132.806,E2 -10132.806} C_VEL
LIN {X 0,Y 421.287,Z 670.085,A -85,B 0,C 180,E1 -10134.276,E2 -10134.276} C_VEL
LIN {X 0,Y 420.454,Z 682.022,A -85,B 0,C 180,E1 -10137.663,E2 -10137.663} C_VEL
LIN {X 0,Y 419.704,Z 694.021,A -85,B 0,C 180,E1 -10140.947,E2 -10140.947} C_VEL
LIN {X 0,Y 419.114,Z 706.077,A -85,B 0,C 180,E1 -10144.152,E2 -10144.152} C_VEL
LIN {X 0,Y 418.561,Z 718.859,A -85,B 0,C 180,E1 -10147.443,E2 -10147.443} C_VEL
LIN {X 0,Y 418.144,Z 733.349,A -85,B 0,C 180,E1 -10151.122,E2 -10151.122} C_VEL
LIN {X 0,Y 417.989,Z 739.311,A -85,B 0,C 180,E1 -10152.614,E2 -10152.614} C_VEL
LIN {X 0,Y 419.554,Z 754.545,A -85,B 0,C 180,E1 -10153.118,E2 -10153.118} C_VEL
LIN {X 0,Y 421.033,Z 772.305,A -85,B 0,C 180,E1 -10153.826,E2 -10153.826} C_VEL
LIN {X 0,Y 421.309,Z 778.843,A -85,B 0,C 180,E1 -10154.147,E2 -10154.147} C_VEL
LIN {X 0,Y 420.72,Z 790.99,A -85,B 0,C 180,E1 -10154.87,E2 -10154.87} C_VEL
LIN {X 0,Y 420.072,Z 802.121,A -85,B 0,C 180,E1 -10155.727,E2 -10155.727} C_VEL
LIN {X 0,Y 419.378,Z 813.139,A -85,B 0,C 180,E1 -10156.801,E2 -10156.801} C_VEL
LIN {X 0,Y 418.842,Z 822.152,A -85,B 0,C 180,E1 -10157.892,E2 -10157.892} C_VEL
LIN {X 0,Y 418.149,Z 831.902,A -85,B 0,C 180,E1 -10159.345,E2 -10159.345} C_VEL
LIN {X 0,Y 417.735,Z 839.656,A -85,B 0,C 180,E1 -10160.803,E2 -10160.803} C_VEL
LIN {X 0,Y 417.415,Z 845.844,A -85,B 0,C 180,E1 -10162.259,E2 -10162.259} C_VEL
LIN {X 0,Y 417.266,Z 850.355,A -85,B 0,C 180,E1 -10163.586,E2 -10163.586} C_VEL
LIN {X 0,Y 417.219,Z 854.474,A -85,B 0,C 180,E1 -10165.168,E2 -10165.168} C_VEL
LIN {X 0,Y 417.104,Z 856.39,A -85,B 0,C 180,E1 -10166.135,E2 -10166.135} C_VEL
LIN {X 0,Y 417.125,Z 857.855,A -85,B 0,C 180,E1 -10167.102,E2 -10167.102} C_VEL
LIN {X 0,Y 417.138,Z 858.875,A -85,B 0,C 180,E1 -10168.068,E2 -10168.068} C_VEL
LIN {X 0,Y 417.115,Z 859.497,A -85,B 0,C 180,E1 -10169.034,E2 -10169.034} C_VEL
LIN {X 0,Y 417.112,Z 859.723,A -85,B 0,C 180,E1 -10169.999,E2 -10169.999} C_VEL
LIN {X 0,Y 417.112,Z 859.502,A -85,B 0,C 180,E1 -10170.965,E2 -10170.965} C_VEL
LIN {X 0,Y 417.135,Z 858.874,A -85,B 0,C 180,E1 -10171.931,E2 -10171.931} C_VEL
LIN {X 0,Y 417.122,Z 857.848,A -85,B 0,C 180,E1 -10172.897,E2 -10172.897} C_VEL
LIN {X 0,Y 417.097,Z 856.399,A -85,B 0,C 180,E1 -10173.864,E2 -10173.864} C_VEL
LIN {X 0,Y 417.213,Z 853.382,A -85,B 0,C 180,E1 -10175.315,E2 -10175.315} C_VEL
LIN {X 0,Y 417.276,Z 849.286,A -85,B 0,C 180,E1 -10176.77,E2 -10176.77} C_VEL
LIN {X 0,Y 417.565,Z 842.968,A -85,B 0,C 180,E1 -10178.468,E2 -10178.468} C_VEL
LIN {X 0,Y 417.935,Z 836.079,A -85,B 0,C 180,E1 -10179.925,E2 -10179.925} C_VEL
LIN {X 0,Y 418.347,Z 829.044,A -85,B 0,C 180,E1 -10181.139,E2 -10181.139} C_VEL
LIN {X 0,Y 418.964,Z 820.546,A -85,B 0,C 180,E1 -10182.349,E2 -10182.349} C_VEL
LIN {X 0,Y 419.609,Z 810.041,A -85,B 0,C 180,E1 -10183.561,E2 -10183.561} C_VEL
LIN {X 0,Y 420.24,Z 799.656,A -85,B 0,C 180,E1 -10184.528,E2 -10184.528} C_VEL
LIN {X 0,Y 420.944,Z 788.245,A -85,B 0,C 180,E1 -10185.369,E2 -10185.369} C_VEL
LIN {X 0,Y 421.493,Z 776.479,A -85,B 0,C 180,E1 -10186.031,E2 -10186.031} C_VEL
LIN {X 0,Y 420.329,Z 763.51,A -85,B 0,C 180,E1 -10186.625,E2 -10186.625} C_VEL
LIN {X 0,Y 418.979,Z 750.125,A -85,B 0,C 180,E1 -10187.035,E2 -10187.035} C_VEL
LIN {X 0,Y 418.009,Z 741.364,A -85,B 0,C 180,E1 -10187.285,E2 -10187.285} C_VEL
LIN {X 0,Y 418.405,Z 728.198,A -85,B 0,C 180,E1 -10190.654,E2 -10190.654} C_VEL
LIN {X 0,Y 419.009,Z 714.313,A -85,B 0,C 180,E1 -10194.263,E2 -10194.263} C_VEL
LIN {X 0,Y 419.647,Z 702.352,A -85,B 0,C 180,E1 -10197.425,E2 -10197.425} C_VEL
LIN {X 0,Y 420.412,Z 689.406,A -85,B 0,C 180,E1 -10200.933,E2 -10200.933} C_VEL
LIN {X 0,Y 421.315,Z 677.426,A -85,B 0,C 180,E1 -10204.261,E2 -10204.261} C_VEL
LIN {X 0,Y 421.94,Z 668.17,A -85,B 0,C 180,E1 -10206.917,E2 -10206.917} C_VEL
LIN {X 0,Y 421.293,Z 663.467,A -85,B 0,C 180,E1 -10208.366,E2 -10208.366} C_VEL
LIN {X 0,Y 419.261,Z 653.226,A -85,B 0,C 180,E1 -10211.691,E2 -10211.691} C_VEL
LIN {X 0,Y 418.225,Z 648.39,A -85,B 0,C 180,E1 -10213.388,E2 -10213.388} C_VEL
LIN {X 0,Y 418.281,Z 648.384,A -85,B 0,C 180,E1 -10216.458,E2 -10216.458} C_VEL
LIN {X 0,Y 418.264,Z 648.383,A -85,B 0,C 180,E1 -10219.122,E2 -10219.122} C_VEL
LIN {X 0,Y 418.236,Z 648.385,A -85,B 0,C 180,E1 -10222.164,E2 -10222.164} C_VEL
LIN {X 0,Y 418.262,Z 648.379,A -85,B 0,C 180,E1 -10225.419,E2 -10225.419} C_VEL
LIN {X 0,Y 418.212,Z 648.387,A -85,B 0,C 180,E1 -10228.604,E2 -10228.604} C_VEL
LIN {X 0,Y 418.291,Z 648.38,A -85,B 0,C 180,E1 -10231.936,E2 -10231.936} C_VEL
LIN {X 0,Y 418.285,Z 648.379,A -85,B 0,C 180,E1 -10235.162,E2 -10235.162} C_VEL
LIN {X 0,Y 418.229,Z 648.387,A -85,B 0,C 180,E1 -10238.303,E2 -10238.303} C_VEL
LIN {X 0,Y 418.279,Z 648.384,A -85,B 0,C 180,E1 -10241.383,E2 -10241.383} C_VEL
LIN {X 0,Y 418.298,Z 648.38,A -85,B 0,C 180,E1 -10244.406,E2 -10244.406} C_VEL
LIN {X 0,Y 418.366,Z 648.371,A -85,B 0,C 180,E1 -10247.386,E2 -10247.386} C_VEL
LIN {X 0,Y 418.356,Z 648.374,A -85,B 0,C 180,E1 -10250.329,E2 -10250.329} C_VEL
LIN {X 0,Y 418.488,Z 648.358,A -85,B 0,C 180,E1 -10253.249,E2 -10253.249} C_VEL
LIN {X 0,Y 418.335,Z 648.376,A -85,B 0,C 180,E1 -10255.181,E2 -10255.181} C_VEL
LIN {X 0,Y 418.539,Z 648.353,A -85,B 0,C 180,E1 -10258.075,E2 -10258.075} C_VEL
LIN {X 0,Y 418.667,Z 648.338,A -85,B 0,C 180,E1 -10260,E2 -10260} C_VEL
LIN {X 0,Y 418.531,Z 648.552,A -85,B 0,C 180,E1 -10261.022,E2 -10261.022} C_VEL
LIN {X 0,Y 419.772,Z 654.921,A -85,B 0,C 180,E1 -10262.879,E2 -10262.879} C_VEL
LIN {X 0,Y 420.506,Z 661.635,A -85,B 0,C 180,E1 -10264.793,E2 -10264.793} C_VEL
LIN {X 0,Y 420.417,Z 672.014,A -85,B 0,C 180,E1 -10267.685,E2 -10267.685} C_VEL
LIN {X 0,Y 420.051,Z 684.161,A -85,B 0,C 180,E1 -10271.093,E2 -10271.093} C_VEL
LIN {X 0,Y 419.689,Z 694.481,A -85,B 0,C 180,E1 -10274.069,E2 -10274.069} C_VEL
LIN {X 0,Y 419.372,Z 705.615,A -85,B 0,C 180,E1 -10277.213,E2 -10277.213} C_VEL
LIN {X 0,Y 418.942,Z 717.425,A -85,B 0,C 180,E1 -10280.627,E2 -10280.627} C_VEL
LIN {X 0,Y 418.613,Z 728.081,A -85,B 0,C 180,E1 -10283.729,E2 -10283.729} C_VEL
LIN {X 0,Y 421.329,Z 741.8,A -85,B 0,C 180,E1 -10284.252,E2 -10284.252} C_VEL
LIN {X 0,Y 422.362,Z 750.129,A -85,B 0,C 180,E1 -10284.647,E2 -10284.647} C_VEL
LIN {X 0,Y 421.832,Z 761.954,A -85,B 0,C 180,E1 -10285.273,E2 -10285.273} C_VEL
LIN {X 0,Y 421.125,Z 773.296,A -85,B 0,C 180,E1 -10286.062,E2 -10286.062} C_VEL
LIN {X 0,Y 420.392,Z 784.523,A -85,B 0,C 180,E1 -10287.057,E2 -10287.057} C_VEL
LIN {X 0,Y 419.612,Z 795.161,A -85,B 0,C 180,E1 -10288.239,E2 -10288.239} C_VEL
LIN {X 0,Y 418.954,Z 804.07,A -85,B 0,C 180,E1 -10289.469,E2 -10289.469} C_VEL
LIN {X 0,Y 418.382,Z 812.188,A -85,B 0,C 180,E1 -10290.841,E2 -10290.841} C_VEL
LIN {X 0,Y 417.932,Z 819.043,A -85,B 0,C 180,E1 -10292.27,E2 -10292.27} C_VEL
LIN {X 0,Y 417.531,Z 824.666,A -85,B 0,C 180,E1 -10293.743,E2 -10293.743} C_VEL
LIN {X 0,Y 417.224,Z 829.731,A -85,B 0,C 180,E1 -10295.485,E2 -10295.485} C_VEL
LIN {X 0,Y 417.007,Z 833.506,A -85,B 0,C 180,E1 -10297.353,E2 -10297.353} C_VEL
LIN {X 0,Y 416.846,Z 835.614,A -85,B 0,C 180,E1 -10299.146,E2 -10299.146} C_VEL
LIN {X 0,Y 416.79,Z 836.358,A -85,B 0,C 180,E1 -10301.119,E2 -10301.119} C_VEL
LIN {X 0,Y 416.802,Z 835.924,A -85,B 0,C 180,E1 -10302.413,E2 -10302.413} C_VEL
LIN {X 0,Y 416.857,Z 834.739,A -85,B 0,C 180,E1 -10303.728,E2 -10303.728} C_VEL
LIN {X 0,Y 416.998,Z 832.774,A -85,B 0,C 180,E1 -10305.061,E2 -10305.061} C_VEL
LIN {X 0,Y 417.159,Z 829.929,A -85,B 0,C 180,E1 -10306.422,E2 -10306.422} C_VEL
LIN {X 0,Y 417.412,Z 826.097,A -85,B 0,C 180,E1 -10307.802,E2 -10307.802} C_VEL
LIN {X 0,Y 417.718,Z 819.971,A -85,B 0,C 180,E1 -10309.488,E2 -10309.488} C_VEL
LIN {X 0,Y 418.284,Z 812.344,A -85,B 0,C 180,E1 -10311.116,E2 -10311.116} C_VEL
LIN {X 0,Y 418.798,Z 804.341,A -85,B 0,C 180,E1 -10312.473,E2 -10312.473} C_VEL
LIN {X 0,Y 419.538,Z 794.387,A -85,B 0,C 180,E1 -10313.839,E2 -10313.839} C_VEL
LIN {X 0,Y 420.28,Z 783.531,A -85,B 0,C 180,E1 -10315.023,E2 -10315.023} C_VEL
LIN {X 0,Y 420.976,Z 772.609,A -85,B 0,C 180,E1 -10315.977,E2 -10315.977} C_VEL
LIN {X 0,Y 421.723,Z 760.615,A -85,B 0,C 180,E1 -10316.792,E2 -10316.792} C_VEL
LIN {X 0,Y 422.225,Z 749.476,A -85,B 0,C 180,E1 -10317.368,E2 -10317.368} C_VEL
LIN {X 0,Y 420.367,Z 737.535,A -85,B 0,C 180,E1 -10317.905,E2 -10317.905} C_VEL
LIN {X 0,Y 418.491,Z 727.646,A -85,B 0,C 180,E1 -10318.258,E2 -10318.258} C_VEL
LIN {X 0,Y 418.986,Z 714.993,A -85,B 0,C 180,E1 -10321.988,E2 -10321.988} C_VEL
LIN {X 0,Y 419.44,Z 702.206,A -85,B 0,C 180,E1 -10325.764,E2 -10325.764} C_VEL
LIN {X 0,Y 419.847,Z 691.554,A -85,B 0,C 180,E1 -10328.907,E2 -10328.907} C_VEL
LIN {X 0,Y 420.218,Z 680.991,A -85,B 0,C 180,E1 -10332.028,E2 -10332.028} C_VEL
LIN {X 0,Y 420.632,Z 669.293,A -85,B 0,C 180,E1 -10335.486,E2 -10335.486} C_VEL
LIN {X 0,Y 420.664,Z 662.681,A -85,B 0,C 180,E1 -10337.457,E2 -10337.457} C_VEL
LIN {X 0,Y 419.874,Z 656.416,A -85,B 0,C 180,E1 -10339.391,E2 -10339.391} C_VEL
LIN {X 0,Y 418.461,Z 648.362,A -85,B 0,C 180,E1 -10341.927,E2 -10341.927} C_VEL
LIN {X 0,Y 418.514,Z 648.358,A -85,B 0,C 180,E1 -10344.218,E2 -10344.218} C_VEL
LIN {X 0,Y 418.322,Z 648.381,A -85,B 0,C 180,E1 -10345.385,E2 -10345.385} C_VEL
LIN {X 0,Y 417.617,Z 648.469,A -85,B 0,C 180,E1 -10346.191,E2 -10346.191} C_VEL
LIN {X 0,Y 414.792,Z 648.821,A -85,B 0,C 180,E1 -10347.501,E2 -10347.501} C_VEL
LIN {X 0,Y 412.493,Z 649.107,A -85,B 0,C 180,E1 -10348.559,E2 -10348.559} C_VEL
LIN {X 0,Y 411.594,Z 649.217,A -85,B 0,C 180,E1 -10349.376,E2 -10349.376} C_VEL
LIN {X 0,Y 411.566,Z 649.22,A -85,B 0,C 180,E1 -10349.651,E2 -10349.651} C_VEL
LIN {X 0,Y 411.468,Z 649.232,A -85,B 0,C 180,E1 -10352.938,E2 -10352.938} C_VEL
LIN {X 0,Y 411.455,Z 649.23,A -85,B 0,C 180,E1 -10356.868,E2 -10356.868} C_VEL
LIN {X 0,Y 411.31,Z 649.248,A -85,B 0,C 180,E1 -10359.839,E2 -10359.839} C_VEL
LIN {X 0,Y 411.315,Z 649.251,A -85,B 0,C 180,E1 -10363.11,E2 -10363.11} C_VEL
LIN {X 0,Y 411.259,Z 649.26,A -85,B 0,C 180,E1 -10366.889,E2 -10366.889} C_VEL
LIN {X 0,Y 411.234,Z 649.263,A -85,B 0,C 180,E1 -10369.987,E2 -10369.987} C_VEL
LIN {X 0,Y 411.248,Z 649.324,A -85,B 0,C 180,E1 -10371.458,E2 -10371.458} C_VEL
LIN {X 0,Y 414.626,Z 660.729,A -85,B 0,C 180,E1 -10372.288,E2 -10372.288} C_VEL
LIN {X 0,Y 415.622,Z 664.786,A -85,B 0,C 180,E1 -10372.625,E2 -10372.625} C_VEL
LIN {X 0,Y 415.084,Z 676.343,A -85,B 0,C 180,E1 -10373.575,E2 -10373.575} C_VEL
LIN {X 0,Y 414.466,Z 686.99,A -85,B 0,C 180,E1 -10374.681,E2 -10374.681} C_VEL
LIN {X 0,Y 413.835,Z 696.988,A -85,B 0,C 180,E1 -10375.967,E2 -10375.967} C_VEL
LIN {X 0,Y 413.19,Z 705.567,A -85,B 0,C 180,E1 -10377.339,E2 -10377.339} C_VEL
LIN {X 0,Y 412.601,Z 712.796,A -85,B 0,C 180,E1 -10378.764,E2 -10378.764} C_VEL
LIN {X 0,Y 412.105,Z 719.731,A -85,B 0,C 180,E1 -10380.488,E2 -10380.488} C_VEL
LIN {X 0,Y 411.779,Z 724.253,A -85,B 0,C 180,E1 -10381.944,E2 -10381.944} C_VEL
LIN {X 0,Y 411.446,Z 728.327,A -85,B 0,C 180,E1 -10383.72,E2 -10383.72} C_VEL
LIN {X 0,Y 411.191,Z 731.067,A -85,B 0,C 180,E1 -10385.53,E2 -10385.53} C_VEL
LIN {X 0,Y 411.135,Z 732.127,A -85,B 0,C 180,E1 -10386.748,E2 -10386.748} C_VEL
LIN {X 0,Y 411.158,Z 732.613,A -85,B 0,C 180,E1 -10388.16,E2 -10388.16} C_VEL
LIN {X 0,Y 411.248,Z 732.187,A -85,B 0,C 180,E1 -10389.734,E2 -10389.734} C_VEL
LIN {X 0,Y 411.401,Z 730.806,A -85,B 0,C 180,E1 -10391.266,E2 -10391.266} C_VEL
LIN {X 0,Y 411.668,Z 727.88,A -85,B 0,C 180,E1 -10393.069,E2 -10393.069} C_VEL
LIN {X 0,Y 411.982,Z 724.849,A -85,B 0,C 180,E1 -10394.381,E2 -10394.381} C_VEL
LIN {X 0,Y 412.462,Z 719.724,A -85,B 0,C 180,E1 -10396.047,E2 -10396.047} C_VEL
LIN {X 0,Y 412.974,Z 714.435,A -85,B 0,C 180,E1 -10397.394,E2 -10397.394} C_VEL
LIN {X 0,Y 413.472,Z 707.775,A -85,B 0,C 180,E1 -10398.776,E2 -10398.776} C_VEL
LIN {X 0,Y 414.186,Z 699.469,A -85,B 0,C 180,E1 -10400.167,E2 -10400.167} C_VEL
LIN {X 0,Y 414.862,Z 690.98,A -85,B 0,C 180,E1 -10401.322,E2 -10401.322} C_VEL
LIN {X 0,Y 415.558,Z 680.327,A -85,B 0,C 180,E1 -10402.495,E2 -10402.495} C_VEL
LIN {X 0,Y 416.182,Z 669.221,A -85,B 0,C 180,E1 -10403.469,E2 -10403.469} C_VEL
LIN {X 0,Y 416.181,Z 665.279,A -85,B 0,C 180,E1 -10403.769,E2 -10403.769} C_VEL
LIN {X 0,Y 412.934,Z 654.47,A -85,B 0,C 180,E1 -10404.643,E2 -10404.643} C_VEL
LIN {X 0,Y 411.226,Z 649.261,A -85,B 0,C 180,E1 -10405.042,E2 -10405.042} C_VEL
LIN {X 0,Y 411.166,Z 649.269,A -85,B 0,C 180,E1 -10408.003,E2 -10408.003} C_VEL
LIN {X 0,Y 411.219,Z 649.261,A -85,B 0,C 180,E1 -10411.41,E2 -10411.41} C_VEL
LIN {X 0,Y 411.237,Z 649.256,A -85,B 0,C 180,E1 -10413.619,E2 -10413.619} C_VEL
LIN {X 0,Y 411.196,Z 649.257,A -85,B 0,C 180,E1 -10416.852,E2 -10416.852} C_VEL
LIN {X 0,Y 411.216,Z 649.264,A -85,B 0,C 180,E1 -10420.051,E2 -10420.051} C_VEL
LIN {X 0,Y 411.266,Z 649.254,A -85,B 0,C 180,E1 -10423.131,E2 -10423.131} C_VEL
LIN {X 0,Y 411.307,Z 649.249,A -85,B 0,C 180,E1 -10426.896,E2 -10426.896} C_VEL
LIN {X 0,Y 411.294,Z 649.254,A -85,B 0,C 180,E1 -10430.161,E2 -10430.161} C_VEL
LIN {X 0,Y 411.483,Z 649.224,A -85,B 0,C 180,E1 -10432.147,E2 -10432.147} C_VEL
LIN {X 0,Y 411.477,Z 649.232,A -85,B 0,C 180,E1 -10434.118,E2 -10434.118} C_VEL
LIN {X 0,Y 411.515,Z 649.224,A -85,B 0,C 180,E1 -10438.043,E2 -10438.043} C_VEL
LIN {X 0,Y 411.644,Z 649.206,A -85,B 0,C 180,E1 -10440,E2 -10440} C_VEL
LIN {X 0,Y 411.468,Z 649.227,A -85,B 0,C 180,E1 -10442.937,E2 -10442.937} C_VEL
LIN {X 0,Y 411.462,Z 649.229,A -85,B 0,C 180,E1 -10446.867,E2 -10446.867} C_VEL
LIN {X 0,Y 411.295,Z 649.246,A -85,B 0,C 180,E1 -10449.839,E2 -10449.839} C_VEL
LIN {X 0,Y 411.307,Z 649.243,A -85,B 0,C 180,E1 -10453.104,E2 -10453.104} C_VEL
LIN {X 0,Y 411.259,Z 649.253,A -85,B 0,C 180,E1 -10456.889,E2 -10456.889} C_VEL
LIN {X 0,Y 411.232,Z 649.257,A -85,B 0,C 180,E1 -10459.987,E2 -10459.987} C_VEL
LIN {X 0,Y 411.205,Z 649.259,A -85,B 0,C 180,E1 -10463.148,E2 -10463.148} C_VEL
LIN {X 0,Y 411.24,Z 649.259,A -85,B 0,C 180,E1 -10466.381,E2 -10466.381} C_VEL
LIN {X 0,Y 411.202,Z 649.262,A -85,B 0,C 180,E1 -10469.713,E2 -10469.713} C_VEL
LIN {X 0,Y 411.208,Z 649.264,A -85,B 0,C 180,E1 -10473.156,E2 -10473.156} C_VEL
LIN {X 0,Y 411.195,Z 649.268,A -85,B 0,C 180,E1 -10476.553,E2 -10476.553} C_VEL
LIN {X 0,Y 411.215,Z 649.263,A -85,B 0,C 180,E1 -10479.728,E2 -10479.728} C_VEL
LIN {X 0,Y 411.176,Z 649.263,A -85,B 0,C 180,E1 -10483.134,E2 -10483.134} C_VEL
LIN {X 0,Y 411.21,Z 649.367,A -85,B 0,C 180,E1 -10486.787,E2 -10486.787} C_VEL
LIN {X 0,Y 413.04,Z 658.207,A -85,B 0,C 180,E1 -10489.969,E2 -10489.969} C_VEL
LIN {X 0,Y 414.534,Z 666.842,A -85,B 0,C 180,E1 -10492.829,E2 -10492.829} C_VEL
LIN {X 0,Y 414.236,Z 672.456,A -85,B 0,C 180,E1 -10494.526,E2 -10494.526} C_VEL
LIN {X 0,Y 413.441,Z 683.15,A -85,B 0,C 180,E1 -10497.624,E2 -10497.624} C_VEL
LIN {X 0,Y 412.647,Z 695.104,A -85,B 0,C 180,E1 -10500.961,E2 -10500.961} C_VEL
LIN {X 0,Y 412.051,Z 707.16,A -85,B 0,C 180,E1 -10504.219,E2 -10504.219} C_VEL
LIN {X 0,Y 411.532,Z 718.665,A -85,B 0,C 180,E1 -10507.249,E2 -10507.249} C_VEL
LIN {X 0,Y 411.094,Z 731.437,A -85,B 0,C 180,E1 -10510.561,E2 -10510.561} C_VEL
LIN {X 0,Y 410.947,Z 738.164,A -85,B 0,C 180,E1 -10512.286,E2 -10512.286} C_VEL
LIN {X 0,Y 412.587,Z 753.603,A -85,B 0,C 180,E1 -10512.815,E2 -10512.815} C_VEL
LIN {X 0,Y 413.967,Z 771.802,A -85,B 0,C 180,E1 -10513.542,E2 -10513.542} C_VEL
LIN {X 0,Y 414.436,Z 778.404,A -85,B 0,C 180,E1 -10513.877,E2 -10513.877} C_VEL
LIN {X 0,Y 413.865,Z 790.608,A -85,B 0,C 180,E1 -10514.613,E2 -10514.613} C_VEL
LIN {X 0,Y 413.135,Z 801.887,A -85,B 0,C 180,E1 -10515.493,E2 -10515.493} C_VEL
LIN {X 0,Y 412.449,Z 812.824,A -85,B 0,C 180,E1 -10516.575,E2 -10516.575} C_VEL
LIN {X 0,Y 411.869,Z 821.855,A -85,B 0,C 180,E1 -10517.684,E2 -10517.684} C_VEL
LIN {X 0,Y 411.132,Z 831.621,A -85,B 0,C 180,E1 -10519.161,E2 -10519.161} C_VEL
LIN {X 0,Y 410.68,Z 839.396,A -85,B 0,C 180,E1 -10520.643,E2 -10520.643} C_VEL
LIN {X 0,Y 410.367,Z 845.598,A -85,B 0,C 180,E1 -10522.125,E2 -10522.125} C_VEL
LIN {X 0,Y 410.193,Z 850.447,A -85,B 0,C 180,E1 -10523.587,E2 -10523.587} C_VEL
LIN {X 0,Y 410.148,Z 854.25,A -85,B 0,C 180,E1 -10525.085,E2 -10525.085} C_VEL
LIN {X 0,Y 410.02,Z 856.17,A -85,B 0,C 180,E1 -10526.068,E2 -10526.068} C_VEL
LIN {X 0,Y 410.022,Z 857.643,A -85,B 0,C 180,E1 -10527.052,E2 -10527.052} C_VEL
LIN {X 0,Y 410.063,Z 858.668,A -85,B 0,C 180,E1 -10528.035,E2 -10528.035} C_VEL
LIN {X 0,Y 410.034,Z 859.293,A -85,B 0,C 180,E1 -10529.017,E2 -10529.017} C_VEL
LIN {X 0,Y 410.029,Z 859.523,A -85,B 0,C 180,E1 -10529.999,E2 -10529.999} C_VEL
LIN {X 0,Y 410.031,Z 859.307,A -85,B 0,C 180,E1 -10530.982,E2 -10530.982} C_VEL
LIN {X 0,Y 410.06,Z 858.681,A -85,B 0,C 180,E1 -10531.964,E2 -10531.964} C_VEL
LIN {X 0,Y 410.019,Z 857.656,A -85,B 0,C 180,E1 -10532.947,E2 -10532.947} C_VEL
LIN {X 0,Y 410.013,Z 856.212,A -85,B 0,C 180,E1 -10533.931,E2 -10533.931} C_VEL
LIN {X 0,Y 410.128,Z 853.197,A -85,B 0,C 180,E1 -10535.407,E2 -10535.407} C_VEL
LIN {X 0,Y 410.199,Z 849.105,A -85,B 0,C 180,E1 -10536.888,E2 -10536.888} C_VEL
LIN {X 0,Y 410.527,Z 842.793,A -85,B 0,C 180,E1 -10538.614,E2 -10538.614} C_VEL
LIN {X 0,Y 410.918,Z 835.921,A -85,B 0,C 180,E1 -10540.096,E2 -10540.096} C_VEL
LIN {X 0,Y 411.338,Z 828.906,A -85,B 0,C 180,E1 -10541.331,E2 -10541.331} C_VEL
LIN {X 0,Y 412.007,Z 820.442,A -85,B 0,C 180,E1 -10542.561,E2 -10542.561} C_VEL
LIN {X 0,Y 412.675,Z 809.969,A -85,B 0,C 180,E1 -10543.793,E2 -10543.793} C_VEL
LIN {X 0,Y 413.452,Z 798.19,A -85,B 0,C 180,E1 -10544.897,E2 -10544.897} C_VEL
LIN {X 0,Y 414.221,Z 786.33,A -85,B 0,C 180,E1 -10545.751,E2 -10545.751} C_VEL
LIN {X 0,Y 414.614,Z 776.609,A -85,B 0,C 180,E1 -10546.304,E2 -10546.304} C_VEL
LIN {X 0,Y 413.533,Z 764.139,A -85,B 0,C 180,E1 -10546.894,E2 -10546.894} C_VEL
LIN {X 0,Y 412.268,Z 750.93,A -85,B 0,C 180,E1 -10547.322,E2 -10547.322} C_VEL
LIN {X 0,Y 410.926,Z 740.305,A -85,B 0,C 180,E1 -10547.611,E2 -10547.611} C_VEL
LIN {X 0,Y 411.384,Z 727.243,A -85,B 0,C 180,E1 -10551.023,E2 -10551.023} C_VEL
LIN {X 0,Y 412.052,Z 713.389,A -85,B 0,C 180,E1 -10554.7,E2 -10554.7} C_VEL
LIN {X 0,Y 412.704,Z 701.134,A -85,B 0,C 180,E1 -10558.019,E2 -10558.019} C_VEL
LIN {X 0,Y 413.48,Z 689.531,A -85,B 0,C 180,E1 -10561.225,E2 -10561.225} C_VEL
LIN {X 0,Y 414.513,Z 676.589,A -85,B 0,C 180,E1 -10564.905,E2 -10564.905} C_VEL
LIN {X 0,Y 414.93,Z 668.648,A -85,B 0,C 180,E1 -10567.243,E2 -10567.243} C_VEL
LIN {X 0,Y 413.698,Z 661.629,A -85,B 0,C 180,E1 -10569.488,E2 -10569.488} C_VEL
LIN {X 0,Y 411.734,Z 651.855,A -85,B 0,C 180,E1 -10572.779,E2 -10572.779} C_VEL
LIN {X 0,Y 411.182,Z 649.268,A -85,B 0,C 180,E1 -10573.739,E2 -10573.739} C_VEL
LIN {X 0,Y 411.228,Z 649.262,A -85,B 0,C 180,E1 -10576.873,E2 -10576.873} C_VEL
LIN {X 0,Y 411.226,Z 649.263,A -85,B 0,C 180,E1 -10580.269,E2 -10580.269} C_VEL
LIN {X 0,Y 411.192,Z 649.263,A -85,B 0,C 180,E1 -10583.446,E2 -10583.446} C_VEL
LIN {X 0,Y 411.203,Z 649.262,A -85,B 0,C 180,E1 -10586.873,E2 -10586.873} C_VEL
LIN {X 0,Y 411.237,Z 649.256,A -85,B 0,C 180,E1 -10590.642,E2 -10590.642} C_VEL
LIN {X 0,Y 411.233,Z 649.259,A -85,B 0,C 180,E1 -10593.619,E2 -10593.619} C_VEL
LIN {X 0,Y 411.199,Z 649.262,A -85,B 0,C 180,E1 -10596.852,E2 -10596.852} C_VEL
LIN {X 0,Y 411.21,Z 649.26,A -85,B 0,C 180,E1 -10600.05,E2 -10600.05} C_VEL
LIN {X 0,Y 411.258,Z 649.257,A -85,B 0,C 180,E1 -10603.131,E2 -10603.131} C_VEL
LIN {X 0,Y 411.309,Z 649.25,A -85,B 0,C 180,E1 -10606.89,E2 -10606.89} C_VEL
LIN {X 0,Y 411.304,Z 649.252,A -85,B 0,C 180,E1 -10610.161,E2 -10610.161} C_VEL
LIN {X 0,Y 411.455,Z 649.234,A -85,B 0,C 180,E1 -10613.133,E2 -10613.133} C_VEL
LIN {X 0,Y 411.306,Z 649.253,A -85,B 0,C 180,E1 -10615.099,E2 -10615.099} C_VEL
LIN {X 0,Y 411.508,Z 649.228,A -85,B 0,C 180,E1 -10618.042,E2 -10618.042} C_VEL
LIN {X 0,Y 411.534,Z 649.279,A -85,B 0,C 180,E1 -10620.581,E2 -10620.581} C_VEL
LIN {X 0,Y 413.016,Z 657.177,A -85,B 0,C 180,E1 -10622.926,E2 -10622.926} C_VEL
LIN {X 0,Y 413.672,Z 663.927,A -85,B 0,C 180,E1 -10624.873,E2 -10624.873} C_VEL
LIN {X 0,Y 413.503,Z 674.347,A -85,B 0,C 180,E1 -10627.815,E2 -10627.815} C_VEL
LIN {X 0,Y 413.058,Z 688.236,A -85,B 0,C 180,E1 -10631.781,E2 -10631.781} C_VEL
LIN {X 0,Y 412.7,Z 698.717,A -85,B 0,C 180,E1 -10634.8,E2 -10634.8} C_VEL
LIN {X 0,Y 412.3,Z 709.362,A -85,B 0,C 180,E1 -10637.868,E2 -10637.868} C_VEL
LIN {X 0,Y 411.9,Z 720.073,A -85,B 0,C 180,E1 -10640.996,E2 -10640.996} C_VEL
LIN {X 0,Y 411.667,Z 728.421,A -85,B 0,C 180,E1 -10643.419,E2 -10643.419} C_VEL
LIN {X 0,Y 414.434,Z 742,A -85,B 0,C 180,E1 -10643.95,E2 -10643.95} C_VEL
LIN {X 0,Y 415.573,Z 750.034,A -85,B 0,C 180,E1 -10644.344,E2 -10644.344} C_VEL
LIN {X 0,Y 415.053,Z 761.877,A -85,B 0,C 180,E1 -10644.977,E2 -10644.977} C_VEL
LIN {X 0,Y 414.265,Z 773.972,A -85,B 0,C 180,E1 -10645.835,E2 -10645.835} C_VEL
LIN {X 0,Y 413.457,Z 785.753,A -85,B 0,C 180,E1 -10646.909,E2 -10646.909} C_VEL
LIN {X 0,Y 412.673,Z 795.812,A -85,B 0,C 180,E1 -10648.066,E2 -10648.066} C_VEL
LIN {X 0,Y 411.993,Z 804.54,A -85,B 0,C 180,E1 -10649.299,E2 -10649.299} C_VEL
LIN {X 0,Y 411.321,Z 813.359,A -85,B 0,C 180,E1 -10650.837,E2 -10650.837} C_VEL
LIN {X 0,Y 410.791,Z 820.868,A -85,B 0,C 180,E1 -10652.511,E2 -10652.511} C_VEL
LIN {X 0,Y 410.46,Z 825.526,A -85,B 0,C 180,E1 -10653.812,E2 -10653.812} C_VEL
LIN {X 0,Y 410.119,Z 830.563,A -85,B 0,C 180,E1 -10655.636,E2 -10655.636} C_VEL
LIN {X 0,Y 409.992,Z 833.015,A -85,B 0,C 180,E1 -10656.867,E2 -10656.867} C_VEL
LIN {X 0,Y 409.854,Z 834.854,A -85,B 0,C 180,E1 -10658.12,E2 -10658.12} C_VEL
LIN {X 0,Y 409.756,Z 836.105,A -85,B 0,C 180,E1 -10659.483,E2 -10659.483} C_VEL
LIN {X 0,Y 409.694,Z 836.569,A -85,B 0,C 180,E1 -10660.995,E2 -10660.995} C_VEL
LIN {X 0,Y 409.719,Z 836.098,A -85,B 0,C 180,E1 -10662.475,E2 -10662.475} C_VEL
LIN {X 0,Y 409.777,Z 834.756,A -85,B 0,C 180,E1 -10663.919,E2 -10663.919} C_VEL
LIN {X 0,Y 409.923,Z 832.571,A -85,B 0,C 180,E1 -10665.338,E2 -10665.338} C_VEL
LIN {X 0,Y 410.104,Z 829.558,A -85,B 0,C 180,E1 -10666.727,E2 -10666.727} C_VEL
LIN {X 0,Y 410.413,Z 824.295,A -85,B 0,C 180,E1 -10668.52,E2 -10668.52} C_VEL
LIN {X 0,Y 410.789,Z 818.936,A -85,B 0,C 180,E1 -10669.919,E2 -10669.919} C_VEL
LIN {X 0,Y 411.292,Z 812.295,A -85,B 0,C 180,E1 -10671.318,E2 -10671.318} C_VEL
LIN {X 0,Y 411.868,Z 804.163,A -85,B 0,C 180,E1 -10672.709,E2 -10672.709} C_VEL
LIN {X 0,Y 412.558,Z 794.85,A -85,B 0,C 180,E1 -10674.006,E2 -10674.006} C_VEL
LIN {X 0,Y 413.303,Z 784.663,A -85,B 0,C 180,E1 -10675.152,E2 -10675.152} C_VEL
LIN {X 0,Y 414.038,Z 773.819,A -85,B 0,C 180,E1 -10676.13,E2 -10676.13} C_VEL
LIN {X 0,Y 414.749,Z 762.365,A -85,B 0,C 180,E1 -10676.947,E2 -10676.947} C_VEL
LIN {X 0,Y 415.355,Z 750.794,A -85,B 0,C 180,E1 -10677.578,E2 -10677.578} C_VEL
LIN {X 0,Y 413.807,Z 740.005,A -85,B 0,C 180,E1 -10678.089,E2 -10678.089} C_VEL
LIN {X 0,Y 411.479,Z 727.843,A -85,B 0,C 180,E1 -10678.529,E2 -10678.529} C_VEL
LIN {X 0,Y 411.988,Z 716.09,A -85,B 0,C 180,E1 -10682.024,E2 -10682.024} C_VEL
LIN {X 0,Y 412.469,Z 703.192,A -85,B 0,C 180,E1 -10685.863,E2 -10685.863} C_VEL
LIN {X 0,Y 412.871,Z 692.476,A -85,B 0,C 180,E1 -10689.056,E2 -10689.056} C_VEL
LIN {X 0,Y 413.266,Z 681.808,A -85,B 0,C 180,E1 -10692.238,E2 -10692.238} C_VEL
LIN {X 0,Y 413.692,Z 670.743,A -85,B 0,C 180,E1 -10695.545,E2 -10695.545} C_VEL
LIN {X 0,Y 413.707,Z 663.476,A -85,B 0,C 180,E1 -10697.741,E2 -10697.741} C_VEL
LIN {X 0,Y 412.828,Z 657.186,A -85,B 0,C 180,E1 -10699.704,E2 -10699.704} C_VEL
LIN {X 0,Y 411.446,Z 649.235,A -85,B 0,C 180,E1 -10702.234,E2 -10702.234} C_VEL
LIN {X 0,Y 411.476,Z 649.236,A -85,B 0,C 180,E1 -10704.119,E2 -10704.119} C_VEL
LIN {X 0,Y 411.515,Z 649.229,A -85,B 0,C 180,E1 -10708.043,E2 -10708.043} C_VEL
LIN {X 0,Y 411.566,Z 649.22,A -85,B 0,C 180,E1 -10709.651,E2 -10709.651} C_VEL
LIN {X 0,Y 411.334,Z 649.25,A -85,B 0,C 180,E1 -10710.197,E2 -10710.197} C_VEL
LIN {X 0,Y 410.022,Z 649.414,A -85,B 0,C 180,E1 -10711.003,E2 -10711.003} C_VEL
LIN {X 0,Y 405.513,Z 649.974,A -85,B 0,C 180,E1 -10712.862,E2 -10712.862} C_VEL
LIN {X 0,Y 404.334,Z 650.118,A -85,B 0,C 180,E1 -10713.691,E2 -10713.691} C_VEL
LIN {X 0,Y 404.205,Z 650.134,A -85,B 0,C 180,E1 -10713.972,E2 -10713.972} C_VEL
LIN {X 0,Y 404.422,Z 650.109,A -85,B 0,C 180,E1 -10715.985,E2 -10715.985} C_VEL
LIN {X 0,Y 404.298,Z 650.123,A -85,B 0,C 180,E1 -10719.001,E2 -10719.001} C_VEL
LIN {X 0,Y 404.272,Z 650.128,A -85,B 0,C 180,E1 -10722.041,E2 -10722.041} C_VEL
LIN {X 0,Y 404.21,Z 650.137,A -85,B 0,C 180,E1 -10725.118,E2 -10725.118} C_VEL
LIN {X 0,Y 404.212,Z 650.138,A -85,B 0,C 180,E1 -10728.238,E2 -10728.238} C_VEL
LIN {X 0,Y 404.188,Z 650.141,A -85,B 0,C 180,E1 -10731.15,E2 -10731.15} C_VEL
LIN {X 0,Y 407.973,Z 662.987,A -85,B 0,C 180,E1 -10732.138,E2 -10732.138} C_VEL
LIN {X 0,Y 408.686,Z 665.589,A -85,B 0,C 180,E1 -10732.363,E2 -10732.363} C_VEL
LIN {X 0,Y 408.35,Z 675.543,A -85,B 0,C 180,E1 -10733.185,E2 -10733.185} C_VEL
LIN {X 0,Y 407.672,Z 686.603,A -85,B 0,C 180,E1 -10734.311,E2 -10734.311} C_VEL
LIN {X 0,Y 407.051,Z 696.495,A -85,B 0,C 180,E1 -10735.572,E2 -10735.572} C_VEL
LIN {X 0,Y 406.372,Z 705.591,A -85,B 0,C 180,E1 -10737,E2 -10737} C_VEL
LIN {X 0,Y 405.723,Z 713.039,A -85,B 0,C 180,E1 -10738.455,E2 -10738.455} C_VEL
LIN {X 0,Y 405.191,Z 720.091,A -85,B 0,C 180,E1 -10740.199,E2 -10740.199} C_VEL
LIN {X 0,Y 404.748,Z 725.848,A -85,B 0,C 180,E1 -10742.091,E2 -10742.091} C_VEL
LIN {X 0,Y 404.435,Z 729.559,A -85,B 0,C 180,E1 -10743.785,E2 -10743.785} C_VEL
LIN {X 0,Y 404.209,Z 731.718,A -85,B 0,C 180,E1 -10745.195,E2 -10745.195} C_VEL
LIN {X 0,Y 404.104,Z 733.218,A -85,B 0,C 180,E1 -10746.869,E2 -10746.869} C_VEL
LIN {X 0,Y 404.168,Z 733.595,A -85,B 0,C 180,E1 -10748.756,E2 -10748.756} C_VEL
LIN {X 0,Y 404.257,Z 732.994,A -85,B 0,C 180,E1 -10750.098,E2 -10750.098} C_VEL
LIN {X 0,Y 404.408,Z 731.435,A -85,B 0,C 180,E1 -10751.645,E2 -10751.645} C_VEL
LIN {X 0,Y 404.706,Z 728.927,A -85,B 0,C 180,E1 -10753.167,E2 -10753.167} C_VEL
LIN {X 0,Y 405.054,Z 725.495,A -85,B 0,C 180,E1 -10754.653,E2 -10754.653} C_VEL
LIN {X 0,Y 405.595,Z 720.27,A -85,B 0,C 180,E1 -10756.345,E2 -10756.345} C_VEL
LIN {X 0,Y 406.166,Z 714.254,A -85,B 0,C 180,E1 -10757.86,E2 -10757.86} C_VEL
LIN {X 0,Y 406.702,Z 708.091,A -85,B 0,C 180,E1 -10759.117,E2 -10759.117} C_VEL
LIN {X 0,Y 407.443,Z 699.819,A -85,B 0,C 180,E1 -10760.498,E2 -10760.498} C_VEL
LIN {X 0,Y 408.158,Z 690.995,A -85,B 0,C 180,E1 -10761.693,E2 -10761.693} C_VEL
LIN {X 0,Y 408.886,Z 680.054,A -85,B 0,C 180,E1 -10762.892,E2 -10762.892} C_VEL
LIN {X 0,Y 409.552,Z 668.542,A -85,B 0,C 180,E1 -10763.883,E2 -10763.883} C_VEL
LIN {X 0,Y 408.774,Z 664.539,A -85,B 0,C 180,E1 -10764.228,E2 -10764.228} C_VEL
LIN {X 0,Y 405.308,Z 653.761,A -85,B 0,C 180,E1 -10765.095,E2 -10765.095} C_VEL
LIN {X 0,Y 404.18,Z 650.14,A -85,B 0,C 180,E1 -10765.363,E2 -10765.363} C_VEL
LIN {X 0,Y 404.143,Z 650.144,A -85,B 0,C 180,E1 -10768.554,E2 -10768.554} C_VEL
LIN {X 0,Y 404.196,Z 650.139,A -85,B 0,C 180,E1 -10772.001,E2 -10772.001} C_VEL
LIN {X 0,Y 404.175,Z 650.14,A -85,B 0,C 180,E1 -10775.334,E2 -10775.334} C_VEL
LIN {X 0,Y 404.139,Z 650.143,A -85,B 0,C 180,E1 -10778.581,E2 -10778.581} C_VEL
LIN {X 0,Y 404.212,Z 650.141,A -85,B 0,C 180,E1 -10781.762,E2 -10781.762} C_VEL
LIN {X 0,Y 404.212,Z 650.133,A -85,B 0,C 180,E1 -10784.882,E2 -10784.882} C_VEL
LIN {X 0,Y 404.257,Z 650.129,A -85,B 0,C 180,E1 -10787.959,E2 -10787.959} C_VEL
LIN {X 0,Y 404.435,Z 650.102,A -85,B 0,C 180,E1 -10792.1,E2 -10792.1} C_VEL
LIN {X 0,Y 404.425,Z 650.109,A -85,B 0,C 180,E1 -10794.015,E2 -10794.015} C_VEL
LIN {X 0,Y 404.484,Z 650.099,A -85,B 0,C 180,E1 -10798.009,E2 -10798.009} C_VEL
LIN {X 0,Y 404.613,Z 650.082,A -85,B 0,C 180,E1 -10800,E2 -10800} C_VEL
LIN {X 0,Y 404.425,Z 650.105,A -85,B 0,C 180,E1 -10802.989,E2 -10802.989} C_VEL
LIN {X 0,Y 404.413,Z 650.107,A -85,B 0,C 180,E1 -10806.987,E2 -10806.987} C_VEL
LIN {X 0,Y 404.26,Z 650.125,A -85,B 0,C 180,E1 -10810.012,E2 -10810.012} C_VEL
LIN {X 0,Y 404.268,Z 650.12,A -85,B 0,C 180,E1 -10813.211,E2 -10813.211} C_VEL
LIN {X 0,Y 404.218,Z 650.13,A -85,B 0,C 180,E1 -10817.007,E2 -10817.007} C_VEL
LIN {X 0,Y 404.166,Z 650.138,A -85,B 0,C 180,E1 -10820.352,E2 -10820.352} C_VEL
LIN {X 0,Y 404.171,Z 650.135,A -85,B 0,C 180,E1 -10823.575,E2 -10823.575} C_VEL
LIN {X 0,Y 404.186,Z 650.134,A -85,B 0,C 180,E1 -10825.767,E2 -10825.767} C_VEL
LIN {X 0,Y 404.197,Z 650.136,A -85,B 0,C 180,E1 -10828,E2 -10828} C_VEL
LIN {X 0,Y 404.141,Z 650.142,A -85,B 0,C 180,E1 -10831.558,E2 -10831.558} C_VEL
LIN {X 0,Y 404.187,Z 650.14,A -85,B 0,C 180,E1 -10835.016,E2 -10835.016} C_VEL
LIN {X 0,Y 404.156,Z 650.146,A -85,B 0,C 180,E1 -10838.757,E2 -10838.757} C_VEL
LIN {X 0,Y 404.125,Z 650.146,A -85,B 0,C 180,E1 -10841.6,E2 -10841.6} C_VEL
LIN {X 0,Y 404.148,Z 650.146,A -85,B 0,C 180,E1 -10844.522,E2 -10844.522} C_VEL
LIN {X 0,Y 404.13,Z 650.215,A -85,B 0,C 180,E1 -10846.378,E2 -10846.378} C_VEL
LIN {X 0,Y 405.699,Z 657.631,A -85,B 0,C 180,E1 -10849.139,E2 -10849.139} C_VEL
LIN {X 0,Y 407.306,Z 666.192,A -85,B 0,C 180,E1 -10852.099,E2 -10852.099} C_VEL
LIN {X 0,Y 407.584,Z 670.542,A -85,B 0,C 180,E1 -10853.495,E2 -10853.495} C_VEL
LIN {X 0,Y 406.582,Z 682.362,A -85,B 0,C 180,E1 -10857.009,E2 -10857.009} C_VEL
LIN {X 0,Y 405.703,Z 694.487,A -85,B 0,C 180,E1 -10860.481,E2 -10860.481} C_VEL
LIN {X 0,Y 405.087,Z 706.22,A -85,B 0,C 180,E1 -10863.742,E2 -10863.742} C_VEL
LIN {X 0,Y 404.494,Z 718.499,A -85,B 0,C 180,E1 -10867.054,E2 -10867.054} C_VEL
LIN {X 0,Y 403.997,Z 732.28,A -85,B 0,C 180,E1 -10870.699,E2 -10870.699} C_VEL
LIN {X 0,Y 403.863,Z 737.006,A -85,B 0,C 180,E1 -10871.942,E2 -10871.942} C_VEL
LIN {X 0,Y 405.707,Z 753.49,A -85,B 0,C 180,E1 -10872.534,E2 -10872.534} C_VEL
LIN {X 0,Y 407.098,Z 772.64,A -85,B 0,C 180,E1 -10873.321,E2 -10873.321} C_VEL
LIN {X 0,Y 407.557,Z 779.034,A -85,B 0,C 180,E1 -10873.662,E2 -10873.662} C_VEL
LIN {X 0,Y 406.864,Z 791.907,A -85,B 0,C 180,E1 -10874.47,E2 -10874.47} C_VEL
LIN {X 0,Y 406.162,Z 802.625,A -85,B 0,C 180,E1 -10875.341,E2 -10875.341} C_VEL
LIN {X 0,Y 405.543,Z 812.362,A -85,B 0,C 180,E1 -10876.328,E2 -10876.328} C_VEL
LIN {X 0,Y 404.908,Z 821.541,A -85,B 0,C 180,E1 -10877.469,E2 -10877.469} C_VEL
LIN {X 0,Y 404.119,Z 831.33,A -85,B 0,C 180,E1 -10878.971,E2 -10878.971} C_VEL
LIN {X 0,Y 403.646,Z 839.134,A -85,B 0,C 180,E1 -10880.479,E2 -10880.479} C_VEL
LIN {X 0,Y 403.31,Z 845.352,A -85,B 0,C 180,E1 -10881.986,E2 -10881.986} C_VEL
LIN {X 0,Y 403.099,Z 850.612,A -85,B 0,C 180,E1 -10883.614,E2 -10883.614} C_VEL
LIN {X 0,Y 403.056,Z 854.025,A -85,B 0,C 180,E1 -10884.998,E2 -10884.998} C_VEL
LIN {X 0,Y 402.939,Z 855.951,A -85,B 0,C 180,E1 -10885.999,E2 -10885.999} C_VEL
LIN {X 0,Y 402.921,Z 857.432,A -85,B 0,C 180,E1 -10887,E2 -10887} C_VEL
LIN {X 0,Y 402.989,Z 858.461,A -85,B 0,C 180,E1 -10888.001,E2 -10888.001} C_VEL
LIN {X 0,Y 402.956,Z 859.09,A -85,B 0,C 180,E1 -10889,E2 -10889} C_VEL
LIN {X 0,Y 402.949,Z 859.323,A -85,B 0,C 180,E1 -10889.999,E2 -10889.999} C_VEL
LIN {X 0,Y 402.953,Z 859.112,A -85,B 0,C 180,E1 -10890.999,E2 -10890.999} C_VEL
LIN {X 0,Y 402.987,Z 858.489,A -85,B 0,C 180,E1 -10891.998,E2 -10891.998} C_VEL
LIN {X 0,Y 402.917,Z 857.467,A -85,B 0,C 180,E1 -10892.999,E2 -10892.999} C_VEL
LIN {X 0,Y 402.931,Z 856.03,A -85,B 0,C 180,E1 -10894,E2 -10894} C_VEL
LIN {X 0,Y 403.024,Z 853.023,A -85,B 0,C 180,E1 -10895.503,E2 -10895.503} C_VEL
LIN {X 0,Y 403.119,Z 848.944,A -85,B 0,C 180,E1 -10897.009,E2 -10897.009} C_VEL
LIN {X 0,Y 403.494,Z 842.649,A -85,B 0,C 180,E1 -10898.766,E2 -10898.766} C_VEL
LIN {X 0,Y 403.907,Z 835.786,A -85,B 0,C 180,E1 -10900.273,E2 -10900.273} C_VEL
LIN {X 0,Y 404.355,Z 828.783,A -85,B 0,C 180,E1 -10901.529,E2 -10901.529} C_VEL
LIN {X 0,Y 405.058,Z 820.342,A -85,B 0,C 180,E1 -10902.78,E2 -10902.78} C_VEL
LIN {X 0,Y 405.767,Z 809.897,A -85,B 0,C 180,E1 -10904.033,E2 -10904.033} C_VEL
LIN {X 0,Y 406.592,Z 798.161,A -85,B 0,C 180,E1 -10905.155,E2 -10905.155} C_VEL
LIN {X 0,Y 407.398,Z 786.373,A -85,B 0,C 180,E1 -10906.022,E2 -10906.022} C_VEL
LIN {X 0,Y 407.764,Z 777.052,A -85,B 0,C 180,E1 -10906.571,E2 -10906.571} C_VEL
LIN {X 0,Y 406.722,Z 764.474,A -85,B 0,C 180,E1 -10907.189,E2 -10907.189} C_VEL
LIN {X 0,Y 405.434,Z 750.856,A -85,B 0,C 180,E1 -10907.651,E2 -10907.651} C_VEL
LIN {X 0,Y 403.868,Z 739.017,A -85,B 0,C 180,E1 -10907.991,E2 -10907.991} C_VEL
LIN {X 0,Y 404.363,Z 726.244,A -85,B 0,C 180,E1 -10911.406,E2 -10911.406} C_VEL
LIN {X 0,Y 405.041,Z 712.68,A -85,B 0,C 180,E1 -10915.092,E2 -10915.092} C_VEL
LIN {X 0,Y 405.731,Z 700.549,A -85,B 0,C 180,E1 -10918.446,E2 -10918.446} C_VEL
LIN {X 0,Y 406.598,Z 689.075,A -85,B 0,C 180,E1 -10921.695,E2 -10921.695} C_VEL
LIN {X 0,Y 407.696,Z 675.72,A -85,B 0,C 180,E1 -10925.576,E2 -10925.576} C_VEL
LIN {X 0,Y 408.024,Z 670.743,A -85,B 0,C 180,E1 -10927.074,E2 -10927.074} C_VEL
LIN {X 0,Y 407.065,Z 664.679,A -85,B 0,C 180,E1 -10929.02,E2 -10929.02} C_VEL
LIN {X 0,Y 405.169,Z 655.087,A -85,B 0,C 180,E1 -10932.272,E2 -10932.272} C_VEL
LIN {X 0,Y 404.149,Z 650.144,A -85,B 0,C 180,E1 -10934.073,E2 -10934.073} C_VEL
LIN {X 0,Y 404.208,Z 650.136,A -85,B 0,C 180,E1 -10937.305,E2 -10937.305} C_VEL
LIN {X 0,Y 404.166,Z 650.141,A -85,B 0,C 180,E1 -10939.955,E2 -10939.955} C_VEL
LIN {X 0,Y 404.138,Z 650.141,A -85,B 0,C 180,E1 -10943.123,E2 -10943.123} C_VEL
LIN {X 0,Y 404.141,Z 650.142,A -85,B 0,C 180,E1 -10946.187,E2 -10946.187} C_VEL
LIN {X 0,Y 404.15,Z 650.143,A -85,B 0,C 180,E1 -10949.715,E2 -10949.715} C_VEL
LIN {X 0,Y 404.191,Z 650.138,A -85,B 0,C 180,E1 -10953.122,E2 -10953.122} C_VEL
LIN {X 0,Y 404.173,Z 650.139,A -85,B 0,C 180,E1 -10955.334,E2 -10955.334} C_VEL
LIN {X 0,Y 404.134,Z 650.144,A -85,B 0,C 180,E1 -10958.58,E2 -10958.58} C_VEL
LIN {X 0,Y 404.205,Z 650.133,A -85,B 0,C 180,E1 -10961.762,E2 -10961.762} C_VEL
LIN {X 0,Y 404.203,Z 650.134,A -85,B 0,C 180,E1 -10964.882,E2 -10964.882} C_VEL
LIN {X 0,Y 404.267,Z 650.127,A -85,B 0,C 180,E1 -10967.959,E2 -10967.959} C_VEL
LIN {X 0,Y 404.428,Z 650.109,A -85,B 0,C 180,E1 -10972.099,E2 -10972.099} C_VEL
LIN {X 0,Y 404.418,Z 650.112,A -85,B 0,C 180,E1 -10974.015,E2 -10974.015} C_VEL
LIN {X 0,Y 404.477,Z 650.104,A -85,B 0,C 180,E1 -10978.008,E2 -10978.008} C_VEL
LIN {X 0,Y 404.563,Z 650.256,A -85,B 0,C 180,E1 -10980.186,E2 -10980.186} C_VEL
LIN {X 0,Y 406.275,Z 659.505,A -85,B 0,C 180,E1 -10982.975,E2 -10982.975} C_VEL
LIN {X 0,Y 406.803,Z 666.265,A -85,B 0,C 180,E1 -10984.955,E2 -10984.955} C_VEL
LIN {X 0,Y 406.586,Z 676.769,A -85,B 0,C 180,E1 -10987.948,E2 -10987.948} C_VEL
LIN {X 0,Y 406.159,Z 688.845,A -85,B 0,C 180,E1 -10991.478,E2 -10991.478} C_VEL
LIN {X 0,Y 405.698,Z 701.298,A -85,B 0,C 180,E1 -10995.061,E2 -10995.061} C_VEL
LIN {X 0,Y 405.218,Z 713.747,A -85,B 0,C 180,E1 -10998.715,E2 -10998.715} C_VEL
LIN {X 0,Y 404.823,Z 724.551,A -85,B 0,C 180,E1 -11001.916,E2 -11001.916} C_VEL
LIN {X 0,Y 404.661,Z 728.458,A -85,B 0,C 180,E1 -11003.074,E2 -11003.074} C_VEL
LIN {X 0,Y 407.421,Z 741.568,A -85,B 0,C 180,E1 -11003.597,E2 -11003.597} C_VEL
LIN {X 0,Y 408.777,Z 752.046,A -85,B 0,C 180,E1 -11004.127,E2 -11004.127} C_VEL
LIN {X 0,Y 408.06,Z 765.174,A -85,B 0,C 180,E1 -11004.89,E2 -11004.89} C_VEL
LIN {X 0,Y 407.283,Z 776.403,A -85,B 0,C 180,E1 -11005.744,E2 -11005.744} C_VEL
LIN {X 0,Y 406.544,Z 786.503,A -85,B 0,C 180,E1 -11006.709,E2 -11006.709} C_VEL
LIN {X 0,Y 405.695,Z 796.831,A -85,B 0,C 180,E1 -11007.936,E2 -11007.936} C_VEL
LIN {X 0,Y 404.961,Z 805.732,A -85,B 0,C 180,E1 -11009.237,E2 -11009.237} C_VEL
LIN {X 0,Y 404.355,Z 813.122,A -85,B 0,C 180,E1 -11010.556,E2 -11010.556} C_VEL
LIN {X 0,Y 403.859,Z 819.931,A -85,B 0,C 180,E1 -11012.056,E2 -11012.056} C_VEL
LIN {X 0,Y 403.356,Z 826.417,A -85,B 0,C 180,E1 -11013.887,E2 -11013.887} C_VEL
LIN {X 0,Y 403.03,Z 831.232,A -85,B 0,C 180,E1 -11015.744,E2 -11015.744} C_VEL
LIN {X 0,Y 402.797,Z 834.536,A -85,B 0,C 180,E1 -11017.639,E2 -11017.639} C_VEL
LIN {X 0,Y 402.68,Z 835.918,A -85,B 0,C 180,E1 -11018.925,E2 -11018.925} C_VEL
LIN {X 0,Y 402.633,Z 836.661,A -85,B 0,C 180,E1 -11020.228,E2 -11020.228} C_VEL
LIN {X 0,Y 402.591,Z 836.678,A -85,B 0,C 180,E1 -11021.557,E2 -11021.557} C_VEL
LIN {X 0,Y 402.645,Z 835.99,A -85,B 0,C 180,E1 -11022.9,E2 -11022.9} C_VEL
LIN {X 0,Y 402.783,Z 833.535,A -85,B 0,C 180,E1 -11024.964,E2 -11024.964} C_VEL
LIN {X 0,Y 402.964,Z 830.625,A -85,B 0,C 180,E1 -11026.453,E2 -11026.453} C_VEL
LIN {X 0,Y 403.308,Z 825.865,A -85,B 0,C 180,E1 -11028.201,E2 -11028.201} C_VEL
LIN {X 0,Y 403.727,Z 819.391,A -85,B 0,C 180,E1 -11029.991,E2 -11029.991} C_VEL
LIN {X 0,Y 404.266,Z 812.509,A -85,B 0,C 180,E1 -11031.472,E2 -11031.472} C_VEL
LIN {X 0,Y 404.936,Z 803.813,A -85,B 0,C 180,E1 -11032.974,E2 -11032.974} C_VEL
LIN {X 0,Y 405.615,Z 794.893,A -85,B 0,C 180,E1 -11034.228,E2 -11034.228} C_VEL
LIN {X 0,Y 406.418,Z 784.414,A -85,B 0,C 180,E1 -11035.416,E2 -11035.416} C_VEL
LIN {X 0,Y 407.242,Z 772.625,A -85,B 0,C 180,E1 -11036.48,E2 -11036.48} C_VEL
LIN {X 0,Y 408.009,Z 760.537,A -85,B 0,C 180,E1 -11037.321,E2 -11037.321} C_VEL
LIN {X 0,Y 408.351,Z 750.08,A -85,B 0,C 180,E1 -11037.886,E2 -11037.886} C_VEL
LIN {X 0,Y 406.185,Z 736.715,A -85,B 0,C 180,E1 -11038.507,E2 -11038.507} C_VEL
LIN {X 0,Y 404.507,Z 727.891,A -85,B 0,C 180,E1 -11038.841,E2 -11038.841} C_VEL
LIN {X 0,Y 405.053,Z 714.977,A -85,B 0,C 180,E1 -11042.722,E2 -11042.722} C_VEL
LIN {X 0,Y 405.557,Z 702.369,A -85,B 0,C 180,E1 -11046.512,E2 -11046.512} C_VEL
LIN {X 0,Y 405.976,Z 691.646,A -85,B 0,C 180,E1 -11049.744,E2 -11049.744} C_VEL
LIN {X 0,Y 406.394,Z 681.16,A -85,B 0,C 180,E1 -11052.904,E2 -11052.904} C_VEL
LIN {X 0,Y 406.775,Z 670.903,A -85,B 0,C 180,E1 -11056.003,E2 -11056.003} C_VEL
LIN {X 0,Y 406.714,Z 664.259,A -85,B 0,C 180,E1 -11058.033,E2 -11058.033} C_VEL
LIN {X 0,Y 405.787,Z 657.959,A -85,B 0,C 180,E1 -11060.027,E2 -11060.027} C_VEL
LIN {X 0,Y 404.39,Z 650.116,A -85,B 0,C 180,E1 -11062.582,E2 -11062.582} C_VEL
LIN {X 0,Y 404.286,Z 650.131,A -85,B 0,C 180,E1 -11065.014,E2 -11065.014} C_VEL
LIN {X 0,Y 404.484,Z 650.105,A -85,B 0,C 180,E1 -11068.009,E2 -11068.009} C_VEL
LIN {X 0,Y 404.613,Z 650.087,A -85,B 0,C 180,E1 -11070.001,E2 -11070.001} C_VEL
LIN {X 0,Y 404.425,Z 650.11,A -85,B 0,C 180,E1 -11072.989,E2 -11072.989} C_VEL
LIN {X 0,Y 404.205,Z 650.134,A -85,B 0,C 180,E1 -11073.972,E2 -11073.972} C_VEL
LIN {X 0,Y 403.483,Z 650.228,A -85,B 0,C 180,E1 -11074.804,E2 -11074.804} C_VEL
LIN {X 0,Y 400.727,Z 650.575,A -85,B 0,C 180,E1 -11076.16,E2 -11076.16} C_VEL
LIN {X 0,Y 398.422,Z 650.861,A -85,B 0,C 180,E1 -11077.255,E2 -11077.255} C_VEL
LIN {X 0,Y 397.403,Z 650.984,A -85,B 0,C 180,E1 -11078.099,E2 -11078.099} C_VEL
LIN {X 0,Y 397.301,Z 650.995,A -85,B 0,C 180,E1 -11078.385,E2 -11078.385} C_VEL
LIN {X 0,Y 397.231,Z 651.005,A -85,B 0,C 180,E1 -11082.258,E2 -11082.258} C_VEL
LIN {X 0,Y 397.182,Z 651.013,A -85,B 0,C 180,E1 -11085.392,E2 -11085.392} C_VEL
LIN {X 0,Y 397.167,Z 651.015,A -85,B 0,C 180,E1 -11088.574,E2 -11088.574} C_VEL
LIN {X 0,Y 397.143,Z 651.02,A -85,B 0,C 180,E1 -11090.864,E2 -11090.864} C_VEL
LIN {X 0,Y 400.95,Z 663.909,A -85,B 0,C 180,E1 -11091.869,E2 -11091.869} C_VEL
LIN {X 0,Y 401.962,Z 667.883,A -85,B 0,C 180,E1 -11092.216,E2 -11092.216} C_VEL
LIN {X 0,Y 401.372,Z 679.191,A -85,B 0,C 180,E1 -11093.202,E2 -11093.202} C_VEL
LIN {X 0,Y 400.699,Z 689.871,A -85,B 0,C 180,E1 -11094.366,E2 -11094.366} C_VEL
LIN {X 0,Y 400.12,Z 698.278,A -85,B 0,C 180,E1 -11095.489,E2 -11095.489} C_VEL
LIN {X 0,Y 399.384,Z 707.336,A -85,B 0,C 180,E1 -11096.965,E2 -11096.965} C_VEL
LIN {X 0,Y 398.742,Z 714.52,A -85,B 0,C 180,E1 -11098.417,E2 -11098.417} C_VEL
LIN {X 0,Y 398.192,Z 721.292,A -85,B 0,C 180,E1 -11100.136,E2 -11100.136} C_VEL
LIN {X 0,Y 397.76,Z 726.867,A -85,B 0,C 180,E1 -11102.01,E2 -11102.01} C_VEL
LIN {X 0,Y 397.409,Z 730.668,A -85,B 0,C 180,E1 -11103.781,E2 -11103.781} C_VEL
LIN {X 0,Y 397.145,Z 733.385,A -85,B 0,C 180,E1 -11105.731,E2 -11105.731} C_VEL
LIN {X 0,Y 397.093,Z 734.428,A -85,B 0,C 180,E1 -11107.209,E2 -11107.209} C_VEL
LIN {X 0,Y 397.15,Z 734.619,A -85,B 0,C 180,E1 -11108.865,E2 -11108.865} C_VEL
LIN {X 0,Y 397.337,Z 733.429,A -85,B 0,C 180,E1 -11110.878,E2 -11110.878} C_VEL
LIN {X 0,Y 397.633,Z 730.729,A -85,B 0,C 180,E1 -11112.881,E2 -11112.881} C_VEL
LIN {X 0,Y 397.975,Z 727.925,A -85,B 0,C 180,E1 -11114.23,E2 -11114.23} C_VEL
LIN {X 0,Y 398.501,Z 723.16,A -85,B 0,C 180,E1 -11115.964,E2 -11115.964} C_VEL
LIN {X 0,Y 399.151,Z 716.825,A -85,B 0,C 180,E1 -11117.69,E2 -11117.69} C_VEL
LIN {X 0,Y 399.736,Z 710.257,A -85,B 0,C 180,E1 -11119.114,E2 -11119.114} C_VEL
LIN {X 0,Y 400.495,Z 702.094,A -85,B 0,C 180,E1 -11120.545,E2 -11120.545} C_VEL
LIN {X 0,Y 401.28,Z 693.331,A -85,B 0,C 180,E1 -11121.791,E2 -11121.791} C_VEL
LIN {X 0,Y 401.967,Z 683.744,A -85,B 0,C 180,E1 -11122.901,E2 -11122.901} C_VEL
LIN {X 0,Y 402.63,Z 673.322,A -85,B 0,C 180,E1 -11123.875,E2 -11123.875} C_VEL
LIN {X 0,Y 402.842,Z 669.601,A -85,B 0,C 180,E1 -11124.175,E2 -11124.175} C_VEL
LIN {X 0,Y 399.615,Z 658.52,A -85,B 0,C 180,E1 -11125.14,E2 -11125.14} C_VEL
LIN {X 0,Y 397.109,Z 651.021,A -85,B 0,C 180,E1 -11125.745,E2 -11125.745} C_VEL
LIN {X 0,Y 397.079,Z 651.025,A -85,B 0,C 180,E1 -11129.118,E2 -11129.118} C_VEL
LIN {X 0,Y 397.195,Z 651.008,A -85,B 0,C 180,E1 -11132.61,E2 -11132.61} C_VEL
LIN {X 0,Y 397.129,Z 651.014,A -85,B 0,C 180,E1 -11135.982,E2 -11135.982} C_VEL
LIN {X 0,Y 397.145,Z 651.019,A -85,B 0,C 180,E1 -11139.703,E2 -11139.703} C_VEL
LIN {X 0,Y 397.185,Z 651.007,A -85,B 0,C 180,E1 -11142.844,E2 -11142.844} C_VEL
LIN {X 0,Y 397.18,Z 651.011,A -85,B 0,C 180,E1 -11145.657,E2 -11145.657} C_VEL
LIN {X 0,Y 397.2,Z 651.002,A -85,B 0,C 180,E1 -11148.777,E2 -11148.777} C_VEL
LIN {X 0,Y 397.396,Z 650.979,A -85,B 0,C 180,E1 -11152.041,E2 -11152.041} C_VEL
LIN {X 0,Y 397.257,Z 650.998,A -85,B 0,C 180,E1 -11154.925,E2 -11154.925} C_VEL
LIN {X 0,Y 397.453,Z 650.974,A -85,B 0,C 180,E1 -11157.973,E2 -11157.973} C_VEL
LIN {X 0,Y 397.582,Z 650.957,A -85,B 0,C 180,E1 -11160,E2 -11160} C_VEL
LIN {X 0,Y 397.383,Z 650.982,A -85,B 0,C 180,E1 -11163.042,E2 -11163.042} C_VEL
LIN {X 0,Y 397.366,Z 650.984,A -85,B 0,C 180,E1 -11167.112,E2 -11167.112} C_VEL
LIN {X 0,Y 397.22,Z 651.004,A -85,B 0,C 180,E1 -11170.191,E2 -11170.191} C_VEL
LIN {X 0,Y 397.228,Z 650.997,A -85,B 0,C 180,E1 -11173.321,E2 -11173.321} C_VEL
LIN {X 0,Y 397.184,Z 651.005,A -85,B 0,C 180,E1 -11177.155,E2 -11177.155} C_VEL
LIN {X 0,Y 397.104,Z 651.02,A -85,B 0,C 180,E1 -11180.73,E2 -11180.73} C_VEL
LIN {X 0,Y 397.135,Z 651.014,A -85,B 0,C 180,E1 -11184.018,E2 -11184.018} C_VEL
LIN {X 0,Y 397.196,Z 651.006,A -85,B 0,C 180,E1 -11187.39,E2 -11187.39} C_VEL
LIN {X 0,Y 397.081,Z 651.024,A -85,B 0,C 180,E1 -11190.883,E2 -11190.883} C_VEL
LIN {X 0,Y 397.127,Z 651.019,A -85,B 0,C 180,E1 -11194.493,E2 -11194.493} C_VEL
LIN {X 0,Y 397.104,Z 651.023,A -85,B 0,C 180,E1 -11198.275,E2 -11198.275} C_VEL
LIN {X 0,Y 397.091,Z 651.024,A -85,B 0,C 180,E1 -11200.909,E2 -11200.909} C_VEL
LIN {X 0,Y 397.103,Z 651.017,A -85,B 0,C 180,E1 -11203.648,E2 -11203.648} C_VEL
LIN {X 0,Y 397.14,Z 651.141,A -85,B 0,C 180,E1 -11205.98,E2 -11205.98} C_VEL
LIN {X 0,Y 398.944,Z 659.915,A -85,B 0,C 180,E1 -11209.321,E2 -11209.321} C_VEL
LIN {X 0,Y 400.424,Z 668.028,A -85,B 0,C 180,E1 -11212.168,E2 -11212.168} C_VEL
LIN {X 0,Y 400.65,Z 671.766,A -85,B 0,C 180,E1 -11213.386,E2 -11213.386} C_VEL
LIN {X 0,Y 399.587,Z 683.495,A -85,B 0,C 180,E1 -11216.959,E2 -11216.959} C_VEL
LIN {X 0,Y 398.627,Z 696.359,A -85,B 0,C 180,E1 -11220.709,E2 -11220.709} C_VEL
LIN {X 0,Y 398.009,Z 707.283,A -85,B 0,C 180,E1 -11223.803,E2 -11223.803} C_VEL
LIN {X 0,Y 397.402,Z 719.29,A -85,B 0,C 180,E1 -11227.103,E2 -11227.103} C_VEL
LIN {X 0,Y 396.907,Z 733.236,A -85,B 0,C 180,E1 -11230.878,E2 -11230.878} C_VEL
LIN {X 0,Y 396.83,Z 735.85,A -85,B 0,C 180,E1 -11231.577,E2 -11231.577} C_VEL
LIN {X 0,Y 398.729,Z 752.647,A -85,B 0,C 180,E1 -11232.207,E2 -11232.207} C_VEL
LIN {X 0,Y 400.226,Z 773.364,A -85,B 0,C 180,E1 -11233.091,E2 -11233.091} C_VEL
LIN {X 0,Y 400.652,Z 779.571,A -85,B 0,C 180,E1 -11233.438,E2 -11233.438} C_VEL
LIN {X 0,Y 400.012,Z 791.407,A -85,B 0,C 180,E1 -11234.197,E2 -11234.197} C_VEL
LIN {X 0,Y 399.255,Z 802.171,A -85,B 0,C 180,E1 -11235.081,E2 -11235.081} C_VEL
LIN {X 0,Y 398.565,Z 812.599,A -85,B 0,C 180,E1 -11236.16,E2 -11236.16} C_VEL
LIN {X 0,Y 397.798,Z 822.968,A -85,B 0,C 180,E1 -11237.5,E2 -11237.5} C_VEL
LIN {X 0,Y 397.106,Z 830.997,A -85,B 0,C 180,E1 -11238.774,E2 -11238.774} C_VEL
LIN {X 0,Y 396.617,Z 838.837,A -85,B 0,C 180,E1 -11240.308,E2 -11240.308} C_VEL
LIN {X 0,Y 396.25,Z 845.074,A -85,B 0,C 180,E1 -11241.842,E2 -11241.842} C_VEL
LIN {X 0,Y 395.994,Z 850.796,A -85,B 0,C 180,E1 -11243.657,E2 -11243.657} C_VEL
LIN {X 0,Y 395.964,Z 853.784,A -85,B 0,C 180,E1 -11244.908,E2 -11244.908} C_VEL
LIN {X 0,Y 395.861,Z 855.717,A -85,B 0,C 180,E1 -11245.927,E2 -11245.927} C_VEL
LIN {X 0,Y 395.82,Z 857.211,A -85,B 0,C 180,E1 -11246.946,E2 -11246.946} C_VEL
LIN {X 0,Y 395.898,Z 858.247,A -85,B 0,C 180,E1 -11247.965,E2 -11247.965} C_VEL
LIN {X 0,Y 395.881,Z 858.882,A -85,B 0,C 180,E1 -11248.982,E2 -11248.982} C_VEL
LIN {X 0,Y 395.871,Z 859.121,A -85,B 0,C 180,E1 -11249.999,E2 -11249.999} C_VEL
LIN {X 0,Y 395.878,Z 858.921,A -85,B 0,C 180,E1 -11251.017,E2 -11251.017} C_VEL
LIN {X 0,Y 395.896,Z 858.303,A -85,B 0,C 180,E1 -11252.034,E2 -11252.034} C_VEL
LIN {X 0,Y 395.816,Z 857.284,A -85,B 0,C 180,E1 -11253.053,E2 -11253.053} C_VEL
LIN {X 0,Y 395.851,Z 855.855,A -85,B 0,C 180,E1 -11254.072,E2 -11254.072} C_VEL
LIN {X 0,Y 395.922,Z 852.856,A -85,B 0,C 180,E1 -11255.602,E2 -11255.602} C_VEL
LIN {X 0,Y 396.063,Z 848.788,A -85,B 0,C 180,E1 -11257.135,E2 -11257.135} C_VEL
LIN {X 0,Y 396.44,Z 842.502,A -85,B 0,C 180,E1 -11258.923,E2 -11258.923} C_VEL
LIN {X 0,Y 396.888,Z 835.65,A -85,B 0,C 180,E1 -11260.457,E2 -11260.457} C_VEL
LIN {X 0,Y 397.384,Z 828.661,A -85,B 0,C 180,E1 -11261.734,E2 -11261.734} C_VEL
LIN {X 0,Y 398.116,Z 820.246,A -85,B 0,C 180,E1 -11263.007,E2 -11263.007} C_VEL
LIN {X 0,Y 398.867,Z 809.859,A -85,B 0,C 180,E1 -11264.28,E2 -11264.28} C_VEL
LIN {X 0,Y 399.75,Z 798.2,A -85,B 0,C 180,E1 -11265.42,E2 -11265.42} C_VEL
LIN {X 0,Y 400.598,Z 786.54,A -85,B 0,C 180,E1 -11266.301,E2 -11266.301} C_VEL
LIN {X 0,Y 400.939,Z 777.751,A -85,B 0,C 180,E1 -11266.84,E2 -11266.84} C_VEL
LIN {X 0,Y 399.999,Z 765.486,A -85,B 0,C 180,E1 -11267.469,E2 -11267.469} C_VEL
LIN {X 0,Y 398.779,Z 752.061,A -85,B 0,C 180,E1 -11267.952,E2 -11267.952} C_VEL
LIN {X 0,Y 396.83,Z 737.9,A -85,B 0,C 180,E1 -11268.388,E2 -11268.388} C_VEL
LIN {X 0,Y 397.326,Z 725.271,A -85,B 0,C 180,E1 -11271.804,E2 -11271.804} C_VEL
LIN {X 0,Y 398.042,Z 712.16,A -85,B 0,C 180,E1 -11275.439,E2 -11275.439} C_VEL
LIN {X 0,Y 398.828,Z 699.645,A -85,B 0,C 180,E1 -11278.985,E2 -11278.985} C_VEL
LIN {X 0,Y 399.806,Z 687.628,A -85,B 0,C 180,E1 -11282.459,E2 -11282.459} C_VEL
LIN {X 0,Y 400.759,Z 676.401,A -85,B 0,C 180,E1 -11285.808,E2 -11285.808} C_VEL
LIN {X 0,Y 400.982,Z 670.83,A -85,B 0,C 180,E1 -11287.521,E2 -11287.521} C_VEL
LIN {X 0,Y 399.241,Z 661.529,A -85,B 0,C 180,E1 -11290.641,E2 -11290.641} C_VEL
LIN {X 0,Y 397.527,Z 653.217,A -85,B 0,C 180,E1 -11293.589,E2 -11293.589} C_VEL
LIN {X 0,Y 397.103,Z 651.021,A -85,B 0,C 180,E1 -11294.409,E2 -11294.409} C_VEL
LIN {X 0,Y 397.158,Z 651.014,A -85,B 0,C 180,E1 -11297.744,E2 -11297.744} C_VEL
LIN {X 0,Y 397.135,Z 651.016,A -85,B 0,C 180,E1 -11301.136,E2 -11301.136} C_VEL
LIN {X 0,Y 397.116,Z 651.016,A -85,B 0,C 180,E1 -11304.496,E2 -11304.496} C_VEL
LIN {X 0,Y 397.076,Z 651.02,A -85,B 0,C 180,E1 -11307.928,E2 -11307.928} C_VEL
LIN {X 0,Y 397.122,Z 651.013,A -85,B 0,C 180,E1 -11311.456,E2 -11311.456} C_VEL
LIN {X 0,Y 397.148,Z 651.009,A -85,B 0,C 180,E1 -11314.487,E2 -11314.487} C_VEL
LIN {X 0,Y 397.104,Z 651.017,A -85,B 0,C 180,E1 -11317.085,E2 -11317.085} C_VEL
LIN {X 0,Y 397.143,Z 651.012,A -85,B 0,C 180,E1 -11320.352,E2 -11320.352} C_VEL
LIN {X 0,Y 397.161,Z 651.014,A -85,B 0,C 180,E1 -11323.553,E2 -11323.553} C_VEL
LIN {X 0,Y 397.223,Z 651.005,A -85,B 0,C 180,E1 -11326.702,E2 -11326.702} C_VEL
LIN {X 0,Y 397.225,Z 651.005,A -85,B 0,C 180,E1 -11329.809,E2 -11329.809} C_VEL
LIN {X 0,Y 397.358,Z 650.989,A -85,B 0,C 180,E1 -11332.888,E2 -11332.888} C_VEL
LIN {X 0,Y 397.25,Z 651.005,A -85,B 0,C 180,E1 -11334.925,E2 -11334.925} C_VEL
LIN {X 0,Y 397.446,Z 650.98,A -85,B 0,C 180,E1 -11337.973,E2 -11337.973} C_VEL
LIN {X 0,Y 397.511,Z 650.996,A -85,B 0,C 180,E1 -11339.683,E2 -11339.683} C_VEL
LIN {X 0,Y 399.293,Z 660.19,A -85,B 0,C 180,E1 -11342.522,E2 -11342.522} C_VEL
LIN {X 0,Y 399.982,Z 666.931,A -85,B 0,C 180,E1 -11344.535,E2 -11344.535} C_VEL
LIN {X 0,Y 399.739,Z 677.426,A -85,B 0,C 180,E1 -11347.577,E2 -11347.577} C_VEL
LIN {X 0,Y 399.304,Z 689.717,A -85,B 0,C 180,E1 -11351.163,E2 -11351.163} C_VEL
LIN {X 0,Y 398.777,Z 702.038,A -85,B 0,C 180,E1 -11354.806,E2 -11354.806} C_VEL
LIN {X 0,Y 398.343,Z 712.966,A -85,B 0,C 180,E1 -11358.028,E2 -11358.028} C_VEL
LIN {X 0,Y 397.884,Z 723.681,A -85,B 0,C 180,E1 -11361.229,E2 -11361.229} C_VEL
LIN {X 0,Y 397.732,Z 728.587,A -85,B 0,C 180,E1 -11362.705,E2 -11362.705} C_VEL
LIN {X 0,Y 400.731,Z 742.84,A -85,B 0,C 180,E1 -11363.316,E2 -11363.316} C_VEL
LIN {X 0,Y 402.047,Z 752.398,A -85,B 0,C 180,E1 -11363.819,E2 -11363.819} C_VEL
LIN {X 0,Y 401.365,Z 764.474,A -85,B 0,C 180,E1 -11364.527,E2 -11364.527} C_VEL
LIN {X 0,Y 400.482,Z 776.707,A -85,B 0,C 180,E1 -11365.464,E2 -11365.464} C_VEL
LIN {X 0,Y 399.608,Z 787.727,A -85,B 0,C 180,E1 -11366.552,E2 -11366.552} C_VEL
LIN {X 0,Y 398.717,Z 798.072,A -85,B 0,C 180,E1 -11367.826,E2 -11367.826} C_VEL
LIN {X 0,Y 398.008,Z 806.18,A -85,B 0,C 180,E1 -11369.051,E2 -11369.051} C_VEL
LIN {X 0,Y 397.273,Z 814.641,A -85,B 0,C 180,E1 -11370.63,E2 -11370.63} C_VEL
LIN {X 0,Y 396.683,Z 822.169,A -85,B 0,C 180,E1 -11372.407,E2 -11372.407} C_VEL
LIN {X 0,Y 396.244,Z 827.475,A -85,B 0,C 180,E1 -11374.033,E2 -11374.033} C_VEL
LIN {X 0,Y 395.921,Z 831.897,A -85,B 0,C 180,E1 -11375.858,E2 -11375.858} C_VEL
LIN {X 0,Y 395.777,Z 834.153,A -85,B 0,C 180,E1 -11377.139,E2 -11377.139} C_VEL
LIN {X 0,Y 395.623,Z 835.905,A -85,B 0,C 180,E1 -11378.591,E2 -11378.591} C_VEL
LIN {X 0,Y 395.538,Z 836.859,A -85,B 0,C 180,E1 -11380.18,E2 -11380.18} C_VEL
LIN {X 0,Y 395.491,Z 836.847,A -85,B 0,C 180,E1 -11381.726,E2 -11381.726} C_VEL
LIN {X 0,Y 395.55,Z 835.928,A -85,B 0,C 180,E1 -11383.243,E2 -11383.243} C_VEL
LIN {X 0,Y 395.723,Z 833.288,A -85,B 0,C 180,E1 -11385.267,E2 -11385.267} C_VEL
LIN {X 0,Y 396.017,Z 829.297,A -85,B 0,C 180,E1 -11387.158,E2 -11387.158} C_VEL
LIN {X 0,Y 396.257,Z 825.208,A -85,B 0,C 180,E1 -11388.578,E2 -11388.578} C_VEL
LIN {X 0,Y 396.663,Z 819.997,A -85,B 0,C 180,E1 -11390.02,E2 -11390.02} C_VEL
LIN {X 0,Y 397.202,Z 813.609,A -85,B 0,C 180,E1 -11391.452,E2 -11391.452} C_VEL
LIN {X 0,Y 397.793,Z 805.723,A -85,B 0,C 180,E1 -11392.887,E2 -11392.887} C_VEL
LIN {X 0,Y 398.522,Z 796.735,A -85,B 0,C 180,E1 -11394.215,E2 -11394.215} C_VEL
LIN {X 0,Y 399.366,Z 786.698,A -85,B 0,C 180,E1 -11395.423,E2 -11395.423} C_VEL
LIN {X 0,Y 400.105,Z 776.625,A -85,B 0,C 180,E1 -11396.407,E2 -11396.407} C_VEL
LIN {X 0,Y 400.907,Z 765.122,A -85,B 0,C 180,E1 -11397.294,E2 -11397.294} C_VEL
LIN {X 0,Y 401.604,Z 751.897,A -85,B 0,C 180,E1 -11398.073,E2 -11398.073} C_VEL
LIN {X 0,Y 399.603,Z 738.947,A -85,B 0,C 180,E1 -11398.71,E2 -11398.71} C_VEL
LIN {X 0,Y 397.483,Z 728.105,A -85,B 0,C 180,E1 -11399.116,E2 -11399.116} C_VEL
LIN {X 0,Y 398.024,Z 716.381,A -85,B 0,C 180,E1 -11402.673,E2 -11402.673} C_VEL
LIN {X 0,Y 398.579,Z 703.844,A -85,B 0,C 180,E1 -11406.477,E2 -11406.477} C_VEL
LIN {X 0,Y 399.043,Z 692.557,A -85,B 0,C 180,E1 -11409.914,E2 -11409.914} C_VEL
LIN {X 0,Y 399.459,Z 682.005,A -85,B 0,C 180,E1 -11413.125,E2 -11413.125} C_VEL
LIN {X 0,Y 399.876,Z 671.705,A -85,B 0,C 180,E1 -11416.275,E2 -11416.275} C_VEL
LIN {X 0,Y 399.731,Z 665.039,A -85,B 0,C 180,E1 -11418.336,E2 -11418.336} C_VEL
LIN {X 0,Y 398.316,Z 656.335,A -85,B 0,C 180,E1 -11421.145,E2 -11421.145} C_VEL
LIN {X 0,Y 397.353,Z 650.993,A -85,B 0,C 180,E1 -11422.889,E2 -11422.889} C_VEL
LIN {X 0,Y 397.257,Z 651.006,A -85,B 0,C 180,E1 -11424.926,E2 -11424.926} C_VEL
LIN {X 0,Y 397.453,Z 650.98,A -85,B 0,C 180,E1 -11427.974,E2 -11427.974} C_VEL
LIN {X 0,Y 397.582,Z 650.963,A -85,B 0,C 180,E1 -11430.001,E2 -11430.001} C_VEL
LIN {X 0,Y 397.383,Z 650.987,A -85,B 0,C 180,E1 -11433.042,E2 -11433.042} C_VEL
LIN {X 0,Y 397.373,Z 650.986,A -85,B 0,C 180,E1 -11436.092,E2 -11436.092} C_VEL
LIN {X 0,Y 397.301,Z 650.995,A -85,B 0,C 180,E1 -11438.385,E2 -11438.385} C_VEL
LIN {X 0,Y 396.576,Z 651.085,A -85,B 0,C 180,E1 -11439.23,E2 -11439.23} C_VEL
LIN {X 0,Y 393.685,Z 651.445,A -85,B 0,C 180,E1 -11440.604,E2 -11440.604} C_VEL
LIN {X 0,Y 391.275,Z 651.747,A -85,B 0,C 180,E1 -11441.714,E2 -11441.714} C_VEL
LIN {X 0,Y 390.252,Z 651.875,A -85,B 0,C 180,E1 -11442.573,E2 -11442.573} C_VEL
LIN {X 0,Y 390.173,Z 651.883,A -85,B 0,C 180,E1 -11442.864,E2 -11442.864} C_VEL
LIN {X 0,Y 390.142,Z 651.889,A -85,B 0,C 180,E1 -11445.677,E2 -11445.677} C_VEL
LIN {X 0,Y 390.111,Z 651.895,A -85,B 0,C 180,E1 -11448.922,E2 -11448.922} C_VEL
LIN {X 0,Y 390.116,Z 651.933,A -85,B 0,C 180,E1 -11450.588,E2 -11450.588} C_VEL
LIN {X 0,Y 393.545,Z 663.461,A -85,B 0,C 180,E1 -11451.475,E2 -11451.475} C_VEL
LIN {X 0,Y 395.138,Z 669.572,A -85,B 0,C 180,E1 -11452.023,E2 -11452.023} C_VEL
LIN {X 0,Y 394.458,Z 681.277,A -85,B 0,C 180,E1 -11453.078,E2 -11453.078} C_VEL
LIN {X 0,Y 393.773,Z 691.567,A -85,B 0,C 180,E1 -11454.237,E2 -11454.237} C_VEL
LIN {X 0,Y 393.165,Z 700.037,A -85,B 0,C 180,E1 -11455.405,E2 -11455.405} C_VEL
LIN {X 0,Y 392.413,Z 708.813,A -85,B 0,C 180,E1 -11456.887,E2 -11456.887} C_VEL
LIN {X 0,Y 391.738,Z 716.361,A -85,B 0,C 180,E1 -11458.468,E2 -11458.468} C_VEL
LIN {X 0,Y 391.161,Z 722.923,A -85,B 0,C 180,E1 -11460.204,E2 -11460.204} C_VEL
LIN {X 0,Y 390.79,Z 727.688,A -85,B 0,C 180,E1 -11461.851,E2 -11461.851} C_VEL
LIN {X 0,Y 390.486,Z 730.908,A -85,B 0,C 180,E1 -11463.295,E2 -11463.295} C_VEL
LIN {X 0,Y 390.18,Z 733.823,A -85,B 0,C 180,E1 -11465.197,E2 -11465.197} C_VEL
LIN {X 0,Y 390.091,Z 735.047,A -85,B 0,C 180,E1 -11466.48,E2 -11466.48} C_VEL
LIN {X 0,Y 390.084,Z 735.611,A -85,B 0,C 180,E1 -11467.776,E2 -11467.776} C_VEL
LIN {X 0,Y 390.165,Z 735.545,A -85,B 0,C 180,E1 -11469.236,E2 -11469.236} C_VEL
LIN {X 0,Y 390.325,Z 734.547,A -85,B 0,C 180,E1 -11470.867,E2 -11470.867} C_VEL
LIN {X 0,Y 390.525,Z 732.635,A -85,B 0,C 180,E1 -11472.452,E2 -11472.452} C_VEL
LIN {X 0,Y 391.057,Z 728.663,A -85,B 0,C 180,E1 -11474.5,E2 -11474.5} C_VEL
LIN {X 0,Y 391.477,Z 724.892,A -85,B 0,C 180,E1 -11475.898,E2 -11475.898} C_VEL
LIN {X 0,Y 392.121,Z 718.996,A -85,B 0,C 180,E1 -11477.612,E2 -11477.612} C_VEL
LIN {X 0,Y 392.906,Z 711.215,A -85,B 0,C 180,E1 -11479.35,E2 -11479.35} C_VEL
LIN {X 0,Y 393.688,Z 703.177,A -85,B 0,C 180,E1 -11480.782,E2 -11480.782} C_VEL
LIN {X 0,Y 394.542,Z 694.172,A -85,B 0,C 180,E1 -11482.081,E2 -11482.081} C_VEL
LIN {X 0,Y 395.3,Z 683.934,A -85,B 0,C 180,E1 -11483.274,E2 -11483.274} C_VEL
LIN {X 0,Y 396.062,Z 672.551,A -85,B 0,C 180,E1 -11484.329,E2 -11484.329} C_VEL
LIN {X 0,Y 395.644,Z 669.166,A -85,B 0,C 180,E1 -11484.629,E2 -11484.629} C_VEL
LIN {X 0,Y 392.112,Z 657.879,A -85,B 0,C 180,E1 -11485.626,E2 -11485.626} C_VEL
LIN {X 0,Y 390.079,Z 651.895,A -85,B 0,C 180,E1 -11486.095,E2 -11486.095} C_VEL
LIN {X 0,Y 390.047,Z 651.901,A -85,B 0,C 180,E1 -11489.869,E2 -11489.869} C_VEL
LIN {X 0,Y 390.114,Z 651.888,A -85,B 0,C 180,E1 -11493.232,E2 -11493.232} C_VEL
LIN {X 0,Y 390.077,Z 651.888,A -85,B 0,C 180,E1 -11496.761,E2 -11496.761} C_VEL
LIN {X 0,Y 390.108,Z 651.893,A -85,B 0,C 180,E1 -11499.983,E2 -11499.983} C_VEL
LIN {X 0,Y 390.143,Z 651.886,A -85,B 0,C 180,E1 -11503.249,E2 -11503.249} C_VEL
LIN {X 0,Y 390.196,Z 651.88,A -85,B 0,C 180,E1 -11506.562,E2 -11506.562} C_VEL
LIN {X 0,Y 390.206,Z 651.877,A -85,B 0,C 180,E1 -11510.671,E2 -11510.671} C_VEL
LIN {X 0,Y 390.32,Z 651.858,A -85,B 0,C 180,E1 -11512.759,E2 -11512.759} C_VEL
LIN {X 0,Y 390.228,Z 651.873,A -85,B 0,C 180,E1 -11514.834,E2 -11514.834} C_VEL
LIN {X 0,Y 390.422,Z 651.849,A -85,B 0,C 180,E1 -11517.937,E2 -11517.937} C_VEL
LIN {X 0,Y 390.552,Z 651.833,A -85,B 0,C 180,E1 -11520,E2 -11520} C_VEL
LIN {X 0,Y 390.317,Z 651.862,A -85,B 0,C 180,E1 -11523.097,E2 -11523.097} C_VEL
LIN {X 0,Y 390.332,Z 651.862,A -85,B 0,C 180,E1 -11526.202,E2 -11526.202} C_VEL
LIN {X 0,Y 390.316,Z 651.861,A -85,B 0,C 180,E1 -11528.282,E2 -11528.282} C_VEL
LIN {X 0,Y 390.173,Z 651.878,A -85,B 0,C 180,E1 -11532.483,E2 -11532.483} C_VEL
LIN {X 0,Y 390.141,Z 651.886,A -85,B 0,C 180,E1 -11535.677,E2 -11535.677} C_VEL
LIN {X 0,Y 390.107,Z 651.888,A -85,B 0,C 180,E1 -11538.922,E2 -11538.922} C_VEL
LIN {X 0,Y 390.042,Z 651.9,A -85,B 0,C 180,E1 -11542.234,E2 -11542.234} C_VEL
LIN {X 0,Y 390.121,Z 651.886,A -85,B 0,C 180,E1 -11545.743,E2 -11545.743} C_VEL
LIN {X 0,Y 390.06,Z 651.897,A -85,B 0,C 180,E1 -11549.11,E2 -11549.11} C_VEL
LIN {X 0,Y 390.045,Z 651.9,A -85,B 0,C 180,E1 -11552.722,E2 -11552.722} C_VEL
LIN {X 0,Y 390.058,Z 651.899,A -85,B 0,C 180,E1 -11555.825,E2 -11555.825} C_VEL
LIN {X 0,Y 390.071,Z 651.898,A -85,B 0,C 180,E1 -11559.218,E2 -11559.218} C_VEL
LIN {X 0,Y 390.045,Z 651.9,A -85,B 0,C 180,E1 -11562.374,E2 -11562.374} C_VEL
LIN {X 0,Y 390.096,Z 652.092,A -85,B 0,C 180,E1 -11565.578,E2 -11565.578} C_VEL
LIN {X 0,Y 391.819,Z 660.545,A -85,B 0,C 180,E1 -11568.882,E2 -11568.882} C_VEL
LIN {X 0,Y 393.354,Z 668.657,A -85,B 0,C 180,E1 -11571.827,E2 -11571.827} C_VEL
LIN {X 0,Y 393.703,Z 672.448,A -85,B 0,C 180,E1 -11573.11,E2 -11573.11} C_VEL
LIN {X 0,Y 392.61,Z 684.499,A -85,B 0,C 180,E1 -11576.866,E2 -11576.866} C_VEL
LIN {X 0,Y 391.635,Z 696.46,A -85,B 0,C 180,E1 -11580.429,E2 -11580.429} C_VEL
LIN {X 0,Y 390.959,Z 707.82,A -85,B 0,C 180,E1 -11583.712,E2 -11583.712} C_VEL
LIN {X 0,Y 390.309,Z 720.282,A -85,B 0,C 180,E1 -11587.223,E2 -11587.223} C_VEL
LIN {X 0,Y 389.77,Z 734.784,A -85,B 0,C 180,E1 -11591.223,E2 -11591.223} C_VEL
LIN {X 0,Y 391.584,Z 749.541,A -85,B 0,C 180,E1 -11591.768,E2 -11591.768} C_VEL
LIN {X 0,Y 392.499,Z 761.75,A -85,B 0,C 180,E1 -11592.294,E2 -11592.294} C_VEL
LIN {X 0,Y 393.383,Z 774.41,A -85,B 0,C 180,E1 -11592.876,E2 -11592.876} C_VEL
LIN {X 0,Y 393.754,Z 780.233,A -85,B 0,C 180,E1 -11593.214,E2 -11593.214} C_VEL
LIN {X 0,Y 393.03,Z 792.645,A -85,B 0,C 180,E1 -11594.042,E2 -11594.042} C_VEL
LIN {X 0,Y 392.263,Z 803.109,A -85,B 0,C 180,E1 -11594.942,E2 -11594.942} C_VEL
LIN {X 0,Y 391.471,Z 813.945,A -85,B 0,C 180,E1 -11596.119,E2 -11596.119} C_VEL
LIN {X 0,Y 390.689,Z 824.379,A -85,B 0,C 180,E1 -11597.533,E2 -11597.533} C_VEL
LIN {X 0,Y 389.894,Z 833.473,A -85,B 0,C 180,E1 -11599.09,E2 -11599.09} C_VEL
LIN {X 0,Y 389.426,Z 840.783,A -85,B 0,C 180,E1 -11600.652,E2 -11600.652} C_VEL
LIN {X 0,Y 389.093,Z 846.607,A -85,B 0,C 180,E1 -11602.214,E2 -11602.214} C_VEL
LIN {X 0,Y 388.865,Z 851.812,A -85,B 0,C 180,E1 -11604.048,E2 -11604.048} C_VEL
LIN {X 0,Y 388.784,Z 855.482,A -85,B 0,C 180,E1 -11605.853,E2 -11605.853} C_VEL
LIN {X 0,Y 388.724,Z 856.988,A -85,B 0,C 180,E1 -11606.89,E2 -11606.89} C_VEL
LIN {X 0,Y 388.794,Z 858.032,A -85,B 0,C 180,E1 -11607.928,E2 -11607.928} C_VEL
LIN {X 0,Y 388.807,Z 858.673,A -85,B 0,C 180,E1 -11608.964,E2 -11608.964} C_VEL
LIN {X 0,Y 388.796,Z 858.918,A -85,B 0,C 180,E1 -11609.999,E2 -11609.999} C_VEL
LIN {X 0,Y 388.805,Z 858.73,A -85,B 0,C 180,E1 -11611.035,E2 -11611.035} C_VEL
LIN {X 0,Y 388.791,Z 858.115,A -85,B 0,C 180,E1 -11612.071,E2 -11612.071} C_VEL
LIN {X 0,Y 388.719,Z 857.101,A -85,B 0,C 180,E1 -11613.109,E2 -11613.109} C_VEL
LIN {X 0,Y 388.774,Z 855.68,A -85,B 0,C 180,E1 -11614.146,E2 -11614.146} C_VEL
LIN {X 0,Y 388.836,Z 852.2,A -85,B 0,C 180,E1 -11615.91,E2 -11615.91} C_VEL
LIN {X 0,Y 389.089,Z 846.998,A -85,B 0,C 180,E1 -11617.785,E2 -11617.785} C_VEL
LIN {X 0,Y 389.442,Z 841.344,A -85,B 0,C 180,E1 -11619.347,E2 -11619.347} C_VEL
LIN {X 0,Y 389.938,Z 834.26,A -85,B 0,C 180,E1 -11620.908,E2 -11620.908} C_VEL
LIN {X 0,Y 390.721,Z 825.41,A -85,B 0,C 180,E1 -11622.465,E2 -11622.465} C_VEL
LIN {X 0,Y 391.411,Z 816.882,A -85,B 0,C 180,E1 -11623.689,E2 -11623.689} C_VEL
LIN {X 0,Y 392.25,Z 806.316,A -85,B 0,C 180,E1 -11624.925,E2 -11624.925} C_VEL
LIN {X 0,Y 393.137,Z 795.217,A -85,B 0,C 180,E1 -11625.953,E2 -11625.953} C_VEL
LIN {X 0,Y 394.019,Z 783.151,A -85,B 0,C 180,E1 -11626.827,E2 -11626.827} C_VEL
LIN {X 0,Y 393.991,Z 777.124,A -85,B 0,C 180,E1 -11627.197,E2 -11627.197} C_VEL
LIN {X 0,Y 393.141,Z 764.626,A -85,B 0,C 180,E1 -11627.839,E2 -11627.839} C_VEL
LIN {X 0,Y 391.857,Z 750.945,A -85,B 0,C 180,E1 -11628.338,E2 -11628.338} C_VEL
LIN {X 0,Y 390.009,Z 738.647,A -85,B 0,C 180,E1 -11628.715,E2 -11628.715} C_VEL
LIN {X 0,Y 389.792,Z 736.162,A -85,B 0,C 180,E1 -11628.884,E2 -11628.884} C_VEL
LIN {X 0,Y 390.306,Z 724.244,A -85,B 0,C 180,E1 -11632.217,E2 -11632.217} C_VEL
LIN {X 0,Y 391.009,Z 712.496,A -85,B 0,C 180,E1 -11635.554,E2 -11635.554} C_VEL
LIN {X 0,Y 391.756,Z 700.673,A -85,B 0,C 180,E1 -11638.971,E2 -11638.971} C_VEL
LIN {X 0,Y 392.781,Z 688.84,A -85,B 0,C 180,E1 -11642.464,E2 -11642.464} C_VEL
LIN {X 0,Y 393.829,Z 676.942,A -85,B 0,C 180,E1 -11646.078,E2 -11646.078} C_VEL
LIN {X 0,Y 394.098,Z 672.948,A -85,B 0,C 180,E1 -11647.323,E2 -11647.323} C_VEL
LIN {X 0,Y 392.633,Z 664.687,A -85,B 0,C 180,E1 -11650.119,E2 -11650.119} C_VEL
LIN {X 0,Y 390.961,Z 656.38,A -85,B 0,C 180,E1 -11653.085,E2 -11653.085} C_VEL
LIN {X 0,Y 390.087,Z 651.896,A -85,B 0,C 180,E1 -11654.792,E2 -11654.792} C_VEL
LIN {X 0,Y 390.103,Z 651.894,A -85,B 0,C 180,E1 -11658.196,E2 -11658.196} C_VEL
LIN {X 0,Y 390.092,Z 651.894,A -85,B 0,C 180,E1 -11660.908,E2 -11660.908} C_VEL
LIN {X 0,Y 390.082,Z 651.89,A -85,B 0,C 180,E1 -11664.793,E2 -11664.793} C_VEL
LIN {X 0,Y 390.023,Z 651.897,A -85,B 0,C 180,E1 -11668.495,E2 -11668.495} C_VEL
LIN {X 0,Y 390.113,Z 651.89,A -85,B 0,C 180,E1 -11672.069,E2 -11672.069} C_VEL
LIN {X 0,Y 390.076,Z 651.897,A -85,B 0,C 180,E1 -11675.519,E2 -11675.519} C_VEL
LIN {X 0,Y 390.051,Z 651.9,A -85,B 0,C 180,E1 -11678.877,E2 -11678.877} C_VEL
LIN {X 0,Y 390.123,Z 651.886,A -85,B 0,C 180,E1 -11682.166,E2 -11682.166} C_VEL
LIN {X 0,Y 390.142,Z 651.887,A -85,B 0,C 180,E1 -11685.392,E2 -11685.392} C_VEL
LIN {X 0,Y 390.156,Z 651.887,A -85,B 0,C 180,E1 -11688.571,E2 -11688.571} C_VEL
LIN {X 0,Y 390.339,Z 651.864,A -85,B 0,C 180,E1 -11691.993,E2 -11691.993} C_VEL
LIN {X 0,Y 390.222,Z 651.879,A -85,B 0,C 180,E1 -11694.833,E2 -11694.833} C_VEL
LIN {X 0,Y 390.415,Z 651.856,A -85,B 0,C 180,E1 -11697.937,E2 -11697.937} C_VEL
LIN {X 0,Y 390.403,Z 652.067,A -85,B 0,C 180,E1 -11699.226,E2 -11699.226} C_VEL
LIN {X 0,Y 391.371,Z 656.099,A -85,B 0,C 180,E1 -11700.514,E2 -11700.514} C_VEL
LIN {X 0,Y 392.8,Z 664.283,A -85,B 0,C 180,E1 -11703.077,E2 -11703.077} C_VEL
LIN {X 0,Y 393.163,Z 669.376,A -85,B 0,C 180,E1 -11704.614,E2 -11704.614} C_VEL
LIN {X 0,Y 392.928,Z 678.153,A -85,B 0,C 180,E1 -11707.192,E2 -11707.192} C_VEL
LIN {X 0,Y 392.404,Z 690.345,A -85,B 0,C 180,E1 -11710.839,E2 -11710.839} C_VEL
LIN {X 0,Y 391.987,Z 700.964,A -85,B 0,C 180,E1 -11713.964,E2 -11713.964} C_VEL
LIN {X 0,Y 391.508,Z 711.872,A -85,B 0,C 180,E1 -11717.229,E2 -11717.229} C_VEL
LIN {X 0,Y 390.964,Z 723.77,A -85,B 0,C 180,E1 -11720.814,E2 -11720.814} C_VEL
LIN {X 0,Y 390.798,Z 728.746,A -85,B 0,C 180,E1 -11722.328,E2 -11722.328} C_VEL
LIN {X 0,Y 393.748,Z 742.683,A -85,B 0,C 180,E1 -11722.947,E2 -11722.947} C_VEL
LIN {X 0,Y 395.28,Z 753.694,A -85,B 0,C 180,E1 -11723.552,E2 -11723.552} C_VEL
LIN {X 0,Y 394.546,Z 765.72,A -85,B 0,C 180,E1 -11724.284,E2 -11724.284} C_VEL
LIN {X 0,Y 393.685,Z 776.881,A -85,B 0,C 180,E1 -11725.162,E2 -11725.162} C_VEL
LIN {X 0,Y 392.794,Z 787.639,A -85,B 0,C 180,E1 -11726.237,E2 -11726.237} C_VEL
LIN {X 0,Y 391.867,Z 797.827,A -85,B 0,C 180,E1 -11727.504,E2 -11727.504} C_VEL
LIN {X 0,Y 391.056,Z 806.594,A -85,B 0,C 180,E1 -11728.846,E2 -11728.846} C_VEL
LIN {X 0,Y 390.355,Z 814.177,A -85,B 0,C 180,E1 -11730.273,E2 -11730.273} C_VEL
LIN {X 0,Y 389.736,Z 821.718,A -85,B 0,C 180,E1 -11732.057,E2 -11732.057} C_VEL
LIN {X 0,Y 389.206,Z 827.552,A -85,B 0,C 180,E1 -11733.838,E2 -11733.838} C_VEL
LIN {X 0,Y 388.873,Z 831.778,A -85,B 0,C 180,E1 -11735.585,E2 -11735.585} C_VEL
LIN {X 0,Y 388.667,Z 834.681,A -85,B 0,C 180,E1 -11737.288,E2 -11737.288} C_VEL
LIN {X 0,Y 388.472,Z 836.676,A -85,B 0,C 180,E1 -11739.286,E2 -11739.286} C_VEL
LIN {X 0,Y 388.418,Z 837.134,A -85,B 0,C 180,E1 -11740.646,E2 -11740.646} C_VEL
LIN {X 0,Y 388.4,Z 836.879,A -85,B 0,C 180,E1 -11742.109,E2 -11742.109} C_VEL
LIN {X 0,Y 388.491,Z 835.75,A -85,B 0,C 180,E1 -11743.647,E2 -11743.647} C_VEL
LIN {X 0,Y 388.693,Z 832.85,A -85,B 0,C 180,E1 -11745.69,E2 -11745.69} C_VEL
LIN {X 0,Y 388.962,Z 829.488,A -85,B 0,C 180,E1 -11747.247,E2 -11747.247} C_VEL
LIN {X 0,Y 389.204,Z 825.324,A -85,B 0,C 180,E1 -11748.716,E2 -11748.716} C_VEL
LIN {X 0,Y 389.645,Z 820.078,A -85,B 0,C 180,E1 -11750.187,E2 -11750.187} C_VEL
LIN {X 0,Y 390.281,Z 812.264,A -85,B 0,C 180,E1 -11751.921,E2 -11751.921} C_VEL
LIN {X 0,Y 391.067,Z 803.484,A -85,B 0,C 180,E1 -11753.467,E2 -11753.467} C_VEL
LIN {X 0,Y 391.861,Z 793.932,A -85,B 0,C 180,E1 -11754.82,E2 -11754.82} C_VEL
LIN {X 0,Y 392.679,Z 783.496,A -85,B 0,C 180,E1 -11756.013,E2 -11756.013} C_VEL
LIN {X 0,Y 393.586,Z 772.014,A -85,B 0,C 180,E1 -11757.061,E2 -11757.061} C_VEL
LIN {X 0,Y 394.418,Z 759.83,A -85,B 0,C 180,E1 -11757.913,E2 -11757.913} C_VEL
LIN {X 0,Y 394.614,Z 751.624,A -85,B 0,C 180,E1 -11758.381,E2 -11758.381} C_VEL
LIN {X 0,Y 392.462,Z 738.3,A -85,B 0,C 180,E1 -11759.045,E2 -11759.045} C_VEL
LIN {X 0,Y 390.518,Z 728.264,A -85,B 0,C 180,E1 -11759.425,E2 -11759.425} C_VEL
LIN {X 0,Y 391.04,Z 717.472,A -85,B 0,C 180,E1 -11762.723,E2 -11762.723} C_VEL
LIN {X 0,Y 391.557,Z 705.93,A -85,B 0,C 180,E1 -11766.261,E2 -11766.261} C_VEL
LIN {X 0,Y 391.999,Z 695.271,A -85,B 0,C 180,E1 -11769.537,E2 -11769.537} C_VEL
LIN {X 0,Y 392.482,Z 684.61,A -85,B 0,C 180,E1 -11772.816,E2 -11772.816} C_VEL
LIN {X 0,Y 392.9,Z 674.197,A -85,B 0,C 180,E1 -11776.027,E2 -11776.027} C_VEL
LIN {X 0,Y 392.893,Z 667.45,A -85,B 0,C 180,E1 -11778.13,E2 -11778.13} C_VEL
LIN {X 0,Y 391.947,Z 660.927,A -85,B 0,C 180,E1 -11780.245,E2 -11780.245} C_VEL
LIN {X 0,Y 390.32,Z 651.868,A -85,B 0,C 180,E1 -11783.279,E2 -11783.279} C_VEL
LIN {X 0,Y 390.422,Z 651.856,A -85,B 0,C 180,E1 -11787.937,E2 -11787.937} C_VEL
LIN {X 0,Y 390.552,Z 651.838,A -85,B 0,C 180,E1 -11790.001,E2 -11790.001} C_VEL
LIN {X 0,Y 390.317,Z 651.868,A -85,B 0,C 180,E1 -11793.097,E2 -11793.097} C_VEL
LIN {X 0,Y 390.327,Z 651.863,A -85,B 0,C 180,E1 -11796.202,E2 -11796.202} C_VEL
LIN {X 0,Y 390.212,Z 651.877,A -85,B 0,C 180,E1 -11799.329,E2 -11799.329} C_VEL
LIN {X 0,Y 390.173,Z 651.883,A -85,B 0,C 180,E1 -11802.864,E2 -11802.864} C_VEL
LIN {X 0,Y 389.513,Z 651.968,A -85,B 0,C 180,E1 -11803.725,E2 -11803.725} C_VEL
LIN {X 0,Y 386.65,Z 652.325,A -85,B 0,C 180,E1 -11805.125,E2 -11805.125} C_VEL
LIN {X 0,Y 384.221,Z 652.627,A -85,B 0,C 180,E1 -11806.256,E2 -11806.256} C_VEL
LIN {X 0,Y 383.18,Z 652.757,A -85,B 0,C 180,E1 -11807.131,E2 -11807.131} C_VEL
LIN {X 0,Y 383.097,Z 652.767,A -85,B 0,C 180,E1 -11807.427,E2 -11807.427} C_VEL
LIN {X 0,Y 383.065,Z 652.773,A -85,B 0,C 180,E1 -11810.261,E2 -11810.261} C_VEL
LIN {X 0,Y 386.914,Z 665.657,A -85,B 0,C 180,E1 -11811.302,E2 -11811.302} C_VEL
LIN {X 0,Y 388.31,Z 670.76,A -85,B 0,C 180,E1 -11811.779,E2 -11811.779} C_VEL
LIN {X 0,Y 387.62,Z 682.75,A -85,B 0,C 180,E1 -11812.887,E2 -11812.887} C_VEL
LIN {X 0,Y 386.874,Z 693.402,A -85,B 0,C 180,E1 -11814.126,E2 -11814.126} C_VEL
LIN {X 0,Y 386.063,Z 703.597,A -85,B 0,C 180,E1 -11815.617,E2 -11815.617} C_VEL
LIN {X 0,Y 385.288,Z 711.971,A -85,B 0,C 180,E1 -11817.131,E2 -11817.131} C_VEL
LIN {X 0,Y 384.645,Z 718.969,A -85,B 0,C 180,E1 -11818.714,E2 -11818.714} C_VEL
LIN {X 0,Y 384.167,Z 724.042,A -85,B 0,C 180,E1 -11820.125,E2 -11820.125} C_VEL
LIN {X 0,Y 383.707,Z 729.467,A -85,B 0,C 180,E1 -11822.085,E2 -11822.085} C_VEL
LIN {X 0,Y 383.444,Z 732.139,A -85,B 0,C 180,E1 -11823.358,E2 -11823.358} C_VEL
LIN {X 0,Y 383.221,Z 734.198,A -85,B 0,C 180,E1 -11824.647,E2 -11824.647} C_VEL
LIN {X 0,Y 383.073,Z 735.823,A -85,B 0,C 180,E1 -11826.173,E2 -11826.173} C_VEL
LIN {X 0,Y 383.061,Z 736.67,A -85,B 0,C 180,E1 -11827.916,E2 -11827.916} C_VEL
LIN {X 0,Y 383.221,Z 736.319,A -85,B 0,C 180,E1 -11829.932,E2 -11829.932} C_VEL
LIN {X 0,Y 383.355,Z 735.247,A -85,B 0,C 180,E1 -11831.299,E2 -11831.299} C_VEL
LIN {X 0,Y 383.744,Z 732.226,A -85,B 0,C 180,E1 -11833.425,E2 -11833.425} C_VEL
LIN {X 0,Y 384.178,Z 729.026,A -85,B 0,C 180,E1 -11834.925,E2 -11834.925} C_VEL
LIN {X 0,Y 384.688,Z 724.895,A -85,B 0,C 180,E1 -11836.411,E2 -11836.411} C_VEL
LIN {X 0,Y 385.272,Z 719.709,A -85,B 0,C 180,E1 -11837.894,E2 -11837.894} C_VEL
LIN {X 0,Y 386.08,Z 712.117,A -85,B 0,C 180,E1 -11839.61,E2 -11839.61} C_VEL
LIN {X 0,Y 386.853,Z 704.645,A -85,B 0,C 180,E1 -11840.969,E2 -11840.969} C_VEL
LIN {X 0,Y 387.651,Z 696.522,A -85,B 0,C 180,E1 -11842.185,E2 -11842.185} C_VEL
LIN {X 0,Y 388.468,Z 687.122,A -85,B 0,C 180,E1 -11843.343,E2 -11843.343} C_VEL
LIN {X 0,Y 389.168,Z 676.977,A -85,B 0,C 180,E1 -11844.357,E2 -11844.357} C_VEL
LIN {X 0,Y 389.373,Z 672.79,A -85,B 0,C 180,E1 -11844.719,E2 -11844.719} C_VEL
LIN {X 0,Y 386.389,Z 662.604,A -85,B 0,C 180,E1 -11845.677,E2 -11845.677} C_VEL
LIN {X 0,Y 383.066,Z 652.769,A -85,B 0,C 180,E1 -11846.489,E2 -11846.489} C_VEL
LIN {X 0,Y 382.993,Z 652.777,A -85,B 0,C 180,E1 -11850.3,E2 -11850.3} C_VEL
LIN {X 0,Y 383.058,Z 652.769,A -85,B 0,C 180,E1 -11852.698,E2 -11852.698} C_VEL
LIN {X 0,Y 383.052,Z 652.769,A -85,B 0,C 180,E1 -11855.04,E2 -11855.04} C_VEL
LIN {X 0,Y 382.996,Z 652.778,A -85,B 0,C 180,E1 -11858.469,E2 -11858.469} C_VEL
LIN {X 0,Y 383.091,Z 652.771,A -85,B 0,C 180,E1 -11861.828,E2 -11861.828} C_VEL
LIN {X 0,Y 383.114,Z 652.763,A -85,B 0,C 180,E1 -11865.119,E2 -11865.119} C_VEL
LIN {X 0,Y 383.098,Z 652.76,A -85,B 0,C 180,E1 -11868.358,E2 -11868.358} C_VEL
LIN {X 0,Y 383.305,Z 652.734,A -85,B 0,C 180,E1 -11871.933,E2 -11871.933} C_VEL
LIN {X 0,Y 383.201,Z 652.749,A -85,B 0,C 180,E1 -11874.739,E2 -11874.739} C_VEL
LIN {X 0,Y 383.389,Z 652.724,A -85,B 0,C 180,E1 -11877.899,E2 -11877.899} C_VEL
LIN {X 0,Y 383.521,Z 652.708,A -85,B 0,C 180,E1 -11880,E2 -11880} C_VEL
LIN {X 0,Y 383.254,Z 652.742,A -85,B 0,C 180,E1 -11883.154,E2 -11883.154} C_VEL
LIN {X 0,Y 383.289,Z 652.74,A -85,B 0,C 180,E1 -11886.316,E2 -11886.316} C_VEL
LIN {X 0,Y 383.262,Z 652.738,A -85,B 0,C 180,E1 -11888.436,E2 -11888.436} C_VEL
LIN {X 0,Y 383.099,Z 652.763,A -85,B 0,C 180,E1 -11891.642,E2 -11891.642} C_VEL
LIN {X 0,Y 383.112,Z 652.761,A -85,B 0,C 180,E1 -11894.882,E2 -11894.882} C_VEL
LIN {X 0,Y 383.091,Z 652.766,A -85,B 0,C 180,E1 -11898.172,E2 -11898.172} C_VEL
LIN {X 0,Y 382.995,Z 652.775,A -85,B 0,C 180,E1 -11901.531,E2 -11901.531} C_VEL
LIN {X 0,Y 383.055,Z 652.768,A -85,B 0,C 180,E1 -11904.96,E2 -11904.96} C_VEL
LIN {X 0,Y 383.019,Z 652.774,A -85,B 0,C 180,E1 -11908.495,E2 -11908.495} C_VEL
LIN {X 0,Y 383.011,Z 652.778,A -85,B 0,C 180,E1 -11912.15,E2 -11912.15} C_VEL
LIN {X 0,Y 383.02,Z 652.776,A -85,B 0,C 180,E1 -11914.668,E2 -11914.668} C_VEL
LIN {X 0,Y 383.001,Z 652.78,A -85,B 0,C 180,E1 -11917.904,E2 -11917.904} C_VEL
LIN {X 0,Y 382.986,Z 652.78,A -85,B 0,C 180,E1 -11921.347,E2 -11921.347} C_VEL
LIN {X 0,Y 383.023,Z 652.776,A -85,B 0,C 180,E1 -11924.949,E2 -11924.949} C_VEL
LIN {X 0,Y 383.288,Z 654.205,A -85,B 0,C 180,E1 -11925.652,E2 -11925.652} C_VEL
LIN {X 0,Y 384.983,Z 662.384,A -85,B 0,C 180,E1 -11928.914,E2 -11928.914} C_VEL
LIN {X 0,Y 386.461,Z 670.243,A -85,B 0,C 180,E1 -11931.807,E2 -11931.807} C_VEL
LIN {X 0,Y 386.748,Z 674.167,A -85,B 0,C 180,E1 -11933.153,E2 -11933.153} C_VEL
LIN {X 0,Y 385.552,Z 686.207,A -85,B 0,C 180,E1 -11936.983,E2 -11936.983} C_VEL
LIN {X 0,Y 384.487,Z 699.303,A -85,B 0,C 180,E1 -11940.952,E2 -11940.952} C_VEL
LIN {X 0,Y 383.738,Z 711.424,A -85,B 0,C 180,E1 -11944.507,E2 -11944.507} C_VEL
LIN {X 0,Y 383.071,Z 723.254,A -85,B 0,C 180,E1 -11947.907,E2 -11947.907} C_VEL
LIN {X 0,Y 382.724,Z 733.691,A -85,B 0,C 180,E1 -11950.838,E2 -11950.838} C_VEL
LIN {X 0,Y 384.539,Z 748.147,A -85,B 0,C 180,E1 -11951.385,E2 -11951.385} C_VEL
LIN {X 0,Y 385.546,Z 760.894,A -85,B 0,C 180,E1 -11951.972,E2 -11951.972} C_VEL
LIN {X 0,Y 386.445,Z 773.935,A -85,B 0,C 180,E1 -11952.571,E2 -11952.571} C_VEL
LIN {X 0,Y 386.827,Z 781.756,A -85,B 0,C 180,E1 -11953.036,E2 -11953.036} C_VEL
LIN {X 0,Y 386.048,Z 793.776,A -85,B 0,C 180,E1 -11953.881,E2 -11953.881} C_VEL
LIN {X 0,Y 385.16,Z 805.232,A -85,B 0,C 180,E1 -11954.928,E2 -11954.928} C_VEL
LIN {X 0,Y 384.402,Z 815.32,A -85,B 0,C 180,E1 -11956.084,E2 -11956.084} C_VEL
LIN {X 0,Y 383.723,Z 824.025,A -85,B 0,C 180,E1 -11957.303,E2 -11957.303} C_VEL
LIN {X 0,Y 382.891,Z 833.153,A -85,B 0,C 180,E1 -11958.887,E2 -11958.887} C_VEL
LIN {X 0,Y 382.396,Z 840.486,A -85,B 0,C 180,E1 -11960.478,E2 -11960.478} C_VEL
LIN {X 0,Y 382.03,Z 846.334,A -85,B 0,C 180,E1 -11962.069,E2 -11962.069} C_VEL
LIN {X 0,Y 381.81,Z 851.033,A -85,B 0,C 180,E1 -11963.713,E2 -11963.713} C_VEL
LIN {X 0,Y 381.771,Z 853.296,A -85,B 0,C 180,E1 -11964.718,E2 -11964.718} C_VEL
LIN {X 0,Y 381.71,Z 855.247,A -85,B 0,C 180,E1 -11965.776,E2 -11965.776} C_VEL
LIN {X 0,Y 381.631,Z 856.764,A -85,B 0,C 180,E1 -11966.832,E2 -11966.832} C_VEL
LIN {X 0,Y 381.691,Z 857.816,A -85,B 0,C 180,E1 -11967.889,E2 -11967.889} C_VEL
LIN {X 0,Y 381.736,Z 858.465,A -85,B 0,C 180,E1 -11968.945,E2 -11968.945} C_VEL
LIN {X 0,Y 381.723,Z 858.715,A -85,B 0,C 180,E1 -11969.999,E2 -11969.999} C_VEL
